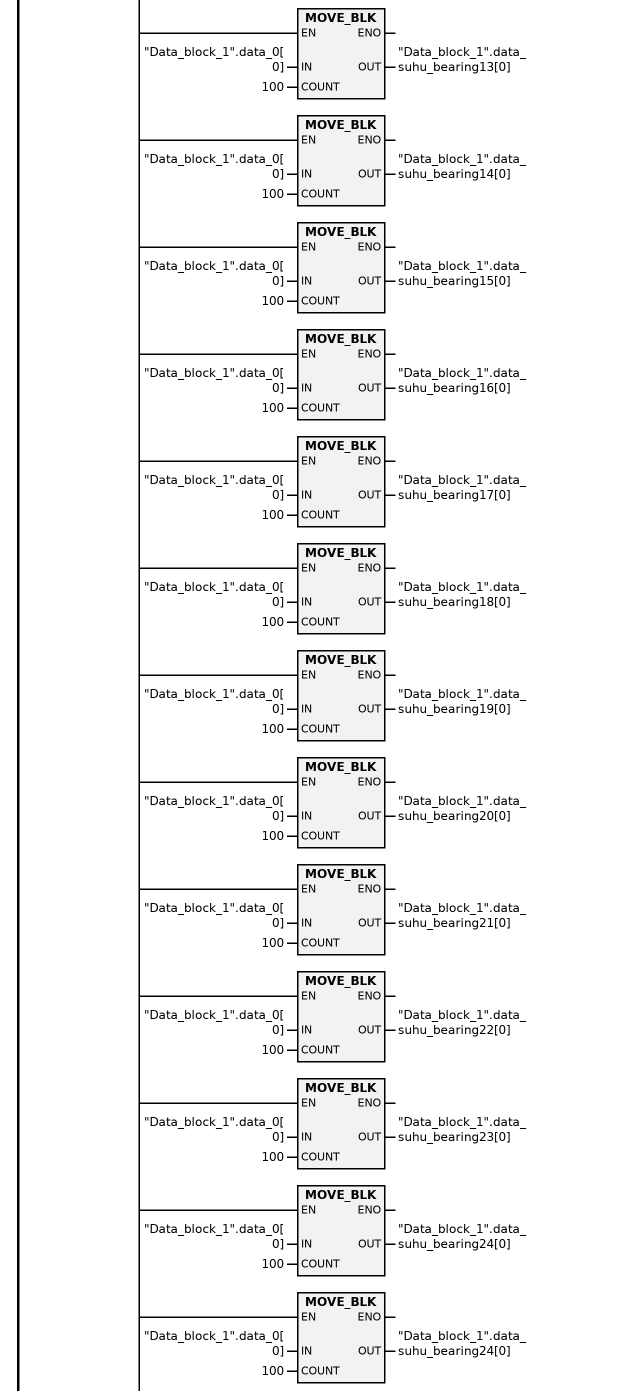
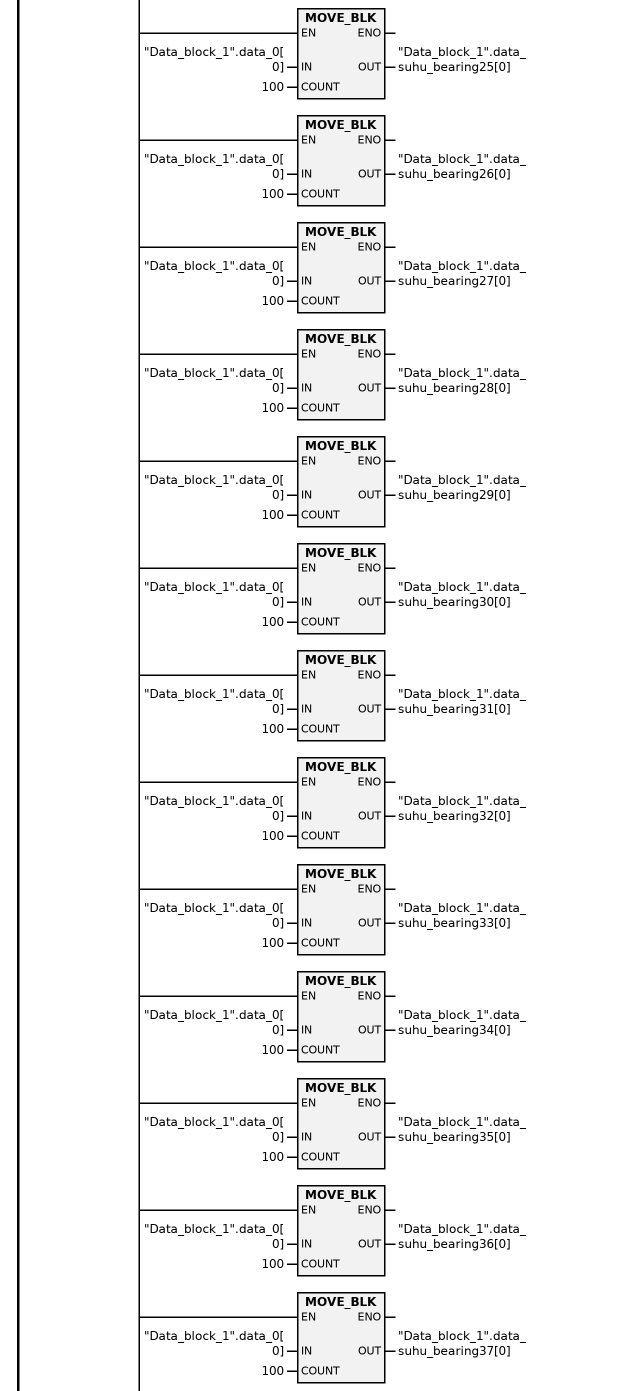
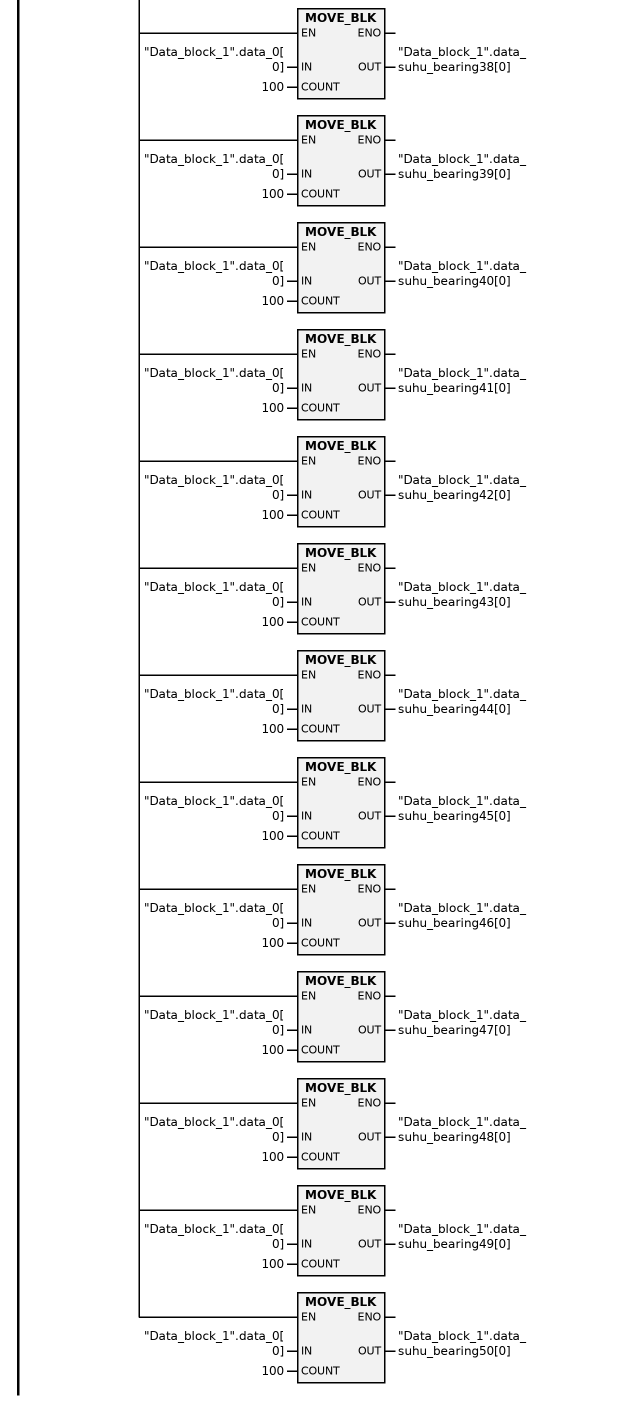
   #_w1 := "Data_block_1".Reset;
   IF #_w1 THEN
       MOVE_BLK(IN := "Data_block_1".data_0[0], COUNT := 100, OUT => "Data_block_1".data_suhu_bearing1[0]);
       MOVE_BLK(IN := "Data_block_1".data_0[0], COUNT := 100, OUT => "Data_block_1".data_suhu_bearing2[0]);
       MOVE_BLK(IN := "Data_block_1".data_0[0], COUNT := 100, OUT => "Data_block_1".data_suhu_bearing3[0]);
       MOVE_BLK(IN := "Data_block_1".data_0[0], COUNT := 100, OUT => "Data_block_1".data_suhu_bearing4[0]);
       MOVE_BLK(IN := "Data_block_1".data_0[0], COUNT := 100, OUT => "Data_block_1".data_suhu_bearing5[0]);
       MOVE_BLK(IN := "Data_block_1".data_0[0], COUNT := 100, OUT => "Data_block_1".data_suhu_bearing6[0]);
       MOVE_BLK(IN := "Data_block_1".data_0[0], COUNT := 100, OUT => "Data_block_1".data_suhu_bearing7[0]);
       MOVE_BLK(IN := "Data_block_1".data_0[0], COUNT := 100, OUT => "Data_block_1".data_suhu_bearing8[0]);
       MOVE_BLK(IN := "Data_block_1".data_0[0], COUNT := 100, OUT => "Data_block_1".data_suhu_bearing9[0]);
       MOVE_BLK(IN := "Data_block_1".data_0[0], COUNT := 100, OUT => "Data_block_1".data_suhu_bearing10[0]);
       MOVE_BLK(IN := "Data_block_1".data_0[0], COUNT := 100, OUT => "Data_block_1".data_suhu_bearing11[0]);
       MOVE_BLK(IN := "Data_block_1".data_0[0], COUNT := 100, OUT => "Data_block_1".data_suhu_bearing12[0]);
       MOVE_BLK(IN := "Data_block_1".data_0[0], COUNT := 100, OUT => "Data_block_1".data_suhu_bearing13[0]);
       MOVE_BLK(IN := "Data_block_1".data_0[0], COUNT := 100, OUT => "Data_block_1".data_suhu_bearing14[0]);
       MOVE_BLK(IN := "Data_block_1".data_0[0], COUNT := 100, OUT => "Data_block_1".data_suhu_bearing15[0]);
       MOVE_BLK(IN := "Data_block_1".data_0[0], COUNT := 100, OUT => "Data_block_1".data_suhu_bearing16[0]);
       MOVE_BLK(IN := "Data_block_1".data_0[0], COUNT := 100, OUT => "Data_block_1".data_suhu_bearing17[0]);
       MOVE_BLK(IN := "Data_block_1".data_0[0], COUNT := 100, OUT => "Data_block_1".data_suhu_bearing18[0]);
       MOVE_BLK(IN := "Data_block_1".data_0[0], COUNT := 100, OUT => "Data_block_1".data_suhu_bearing19[0]);
       MOVE_BLK(IN := "Data_block_1".data_0[0], COUNT := 100, OUT => "Data_block_1".data_suhu_bearing20[0]);
       MOVE_BLK(IN := "Data_block_1".data_0[0], COUNT := 100, OUT => "Data_block_1".data_suhu_bearing21[0]);
       MOVE_BLK(IN := "Data_block_1".data_0[0], COUNT := 100, OUT => "Data_block_1".data_suhu_bearing22[0]);
       MOVE_BLK(IN := "Data_block_1".data_0[0], COUNT := 100, OUT => "Data_block_1".data_suhu_bearing23[0]);
       MOVE_BLK(IN := "Data_block_1".data_0[0], COUNT := 100, OUT => "Data_block_1".data_suhu_bearing24[0]);
       MOVE_BLK(IN := "Data_block_1".data_0[0], COUNT := 100, OUT => "Data_block_1".data_suhu_bearing24[0]);
       MOVE_BLK(IN := "Data_block_1".data_0[0], COUNT := 100, OUT => "Data_block_1".data_suhu_bearing25[0]);
       MOVE_BLK(IN := "Data_block_1".data_0[0], COUNT := 100, OUT => "Data_block_1".data_suhu_bearing26[0]);
       MOVE_BLK(IN := "Data_block_1".data_0[0], COUNT := 100, OUT => "Data_block_1".data_suhu_bearing27[0]);
       MOVE_BLK(IN := "Data_block_1".data_0[0], COUNT := 100, OUT => "Data_block_1".data_suhu_bearing28[0]);
       MOVE_BLK(IN := "Data_block_1".data_0[0], COUNT := 100, OUT => "Data_block_1".data_suhu_bearing29[0]);
       MOVE_BLK(IN := "Data_block_1".data_0[0], COUNT := 100, OUT => "Data_block_1".data_suhu_bearing30[0]);
       MOVE_BLK(IN := "Data_block_1".data_0[0], COUNT := 100, OUT => "Data_block_1".data_suhu_bearing31[0]);
       MOVE_BLK(IN := "Data_block_1".data_0[0], COUNT := 100, OUT => "Data_block_1".data_suhu_bearing32[0]);
       MOVE_BLK(IN := "Data_block_1".data_0[0], COUNT := 100, OUT => "Data_block_1".data_suhu_bearing33[0]);
       MOVE_BLK(IN := "Data_block_1".data_0[0], COUNT := 100, OUT => "Data_block_1".data_suhu_bearing34[0]);
       MOVE_BLK(IN := "Data_block_1".data_0[0], COUNT := 100, OUT => "Data_block_1".data_suhu_bearing35[0]);
       MOVE_BLK(IN := "Data_block_1".data_0[0], COUNT := 100, OUT => "Data_block_1".data_suhu_bearing36[0]);
       MOVE_BLK(IN := "Data_block_1".data_0[0], COUNT := 100, OUT => "Data_block_1".data_suhu_bearing37[0]);
       MOVE_BLK(IN := "Data_block_1".data_0[0], COUNT := 100, OUT => "Data_block_1".data_suhu_bearing38[0]);
       MOVE_BLK(IN := "Data_block_1".data_0[0], COUNT := 100, OUT => "Data_block_1".data_suhu_bearing39[0]);
       MOVE_BLK(IN := "Data_block_1".data_0[0], COUNT := 100, OUT => "Data_block_1".data_suhu_bearing40[0]);
       MOVE_BLK(IN := "Data_block_1".data_0[0], COUNT := 100, OUT => "Data_block_1".data_suhu_bearing41[0]);
       MOVE_BLK(IN := "Data_block_1".data_0[0], COUNT := 100, OUT => "Data_block_1".data_suhu_bearing42[0]);
       MOVE_BLK(IN := "Data_block_1".data_0[0], COUNT := 100, OUT => "Data_block_1".data_suhu_bearing43[0]);
       MOVE_BLK(IN := "Data_block_1".data_0[0], COUNT := 100, OUT => "Data_block_1".data_suhu_bearing44[0]);
       MOVE_BLK(IN := "Data_block_1".data_0[0], COUNT := 100, OUT => "Data_block_1".data_suhu_bearing45[0]);
       MOVE_BLK(IN := "Data_block_1".data_0[0], COUNT := 100, OUT => "Data_block_1".data_suhu_bearing46[0]);
       MOVE_BLK(IN := "Data_block_1".data_0[0], COUNT := 100, OUT => "Data_block_1".data_suhu_bearing47[0]);
       MOVE_BLK(IN := "Data_block_1".data_0[0], COUNT := 100, OUT => "Data_block_1".data_suhu_bearing48[0]);
       MOVE_BLK(IN := "Data_block_1".data_0[0], COUNT := 100, OUT => "Data_block_1".data_suhu_bearing49[0]);
       MOVE_BLK(IN := "Data_block_1".data_0[0], COUNT := 100, OUT => "Data_block_1".data_suhu_bearing50[0]);
   END_IF;
END_REGION

REGION Network 24: Mengukur Suhu Roda (kiri ke kanan)
   // setelah sensor suhu aktif membaca
   // kemudian counter menghitung jumlah berapa kali sensor suhu mendeteksi suhu pada satu roda
   // 
   // apabila data sensor suhu yang terbaca(datasensor) tidak sama dengan nol maka data suhu yang terbaca(datasensor) dipindahkan ke array data suhu baru (data_baru1 untuk sebelah kanan) (data_baru2 untuk sebelah kiri)
   // data sensor terbaru dirubah jadi data baru
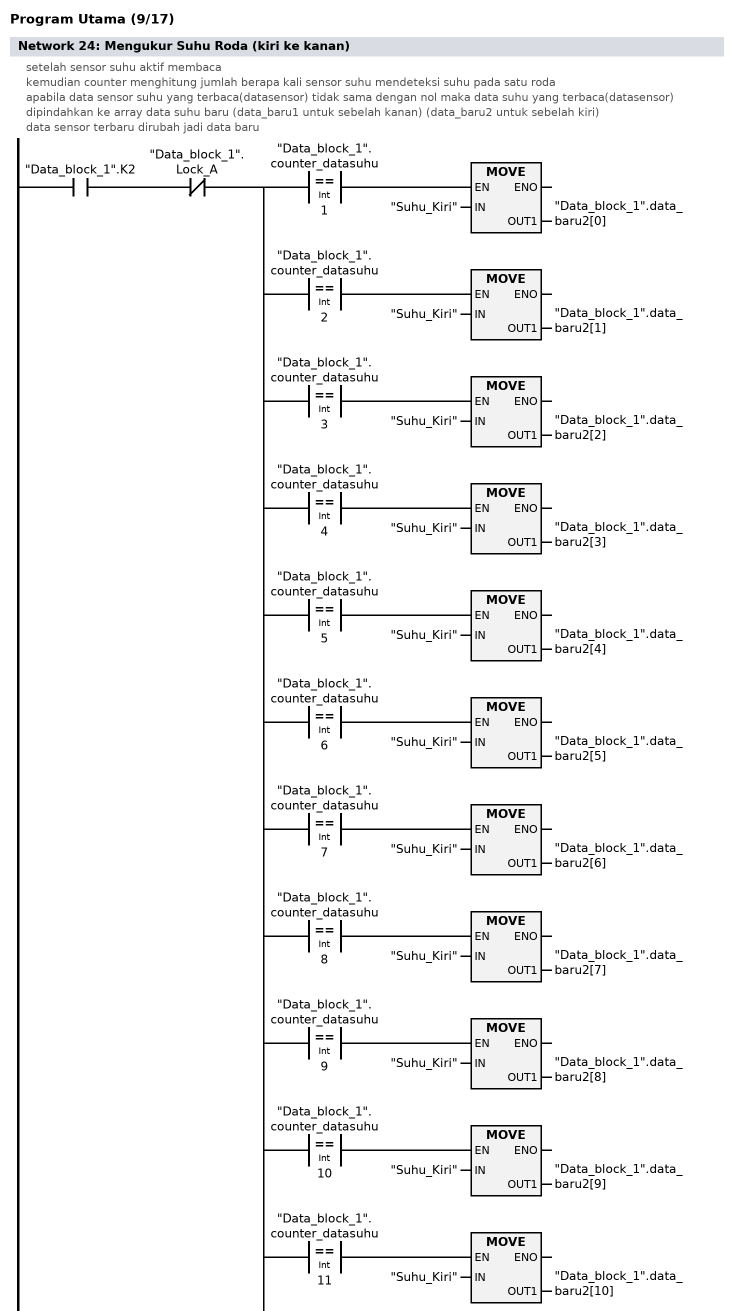
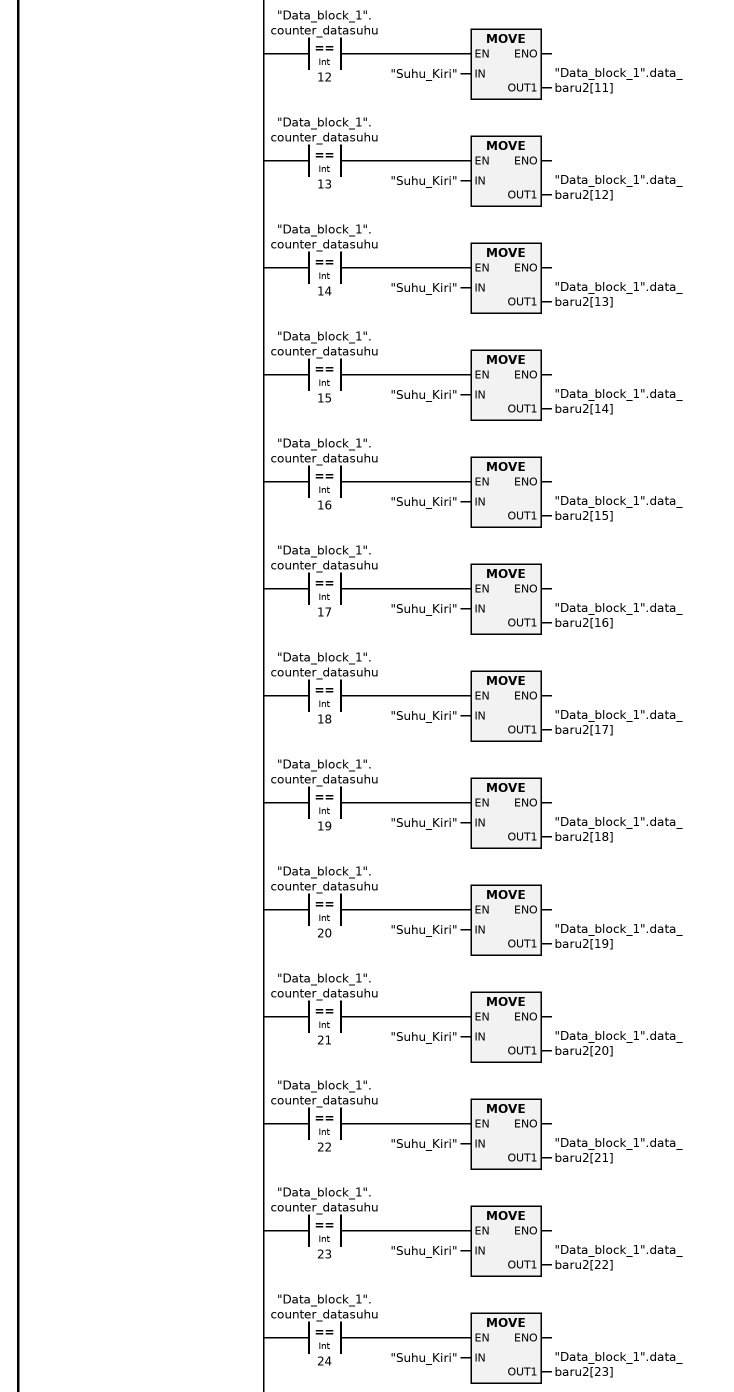
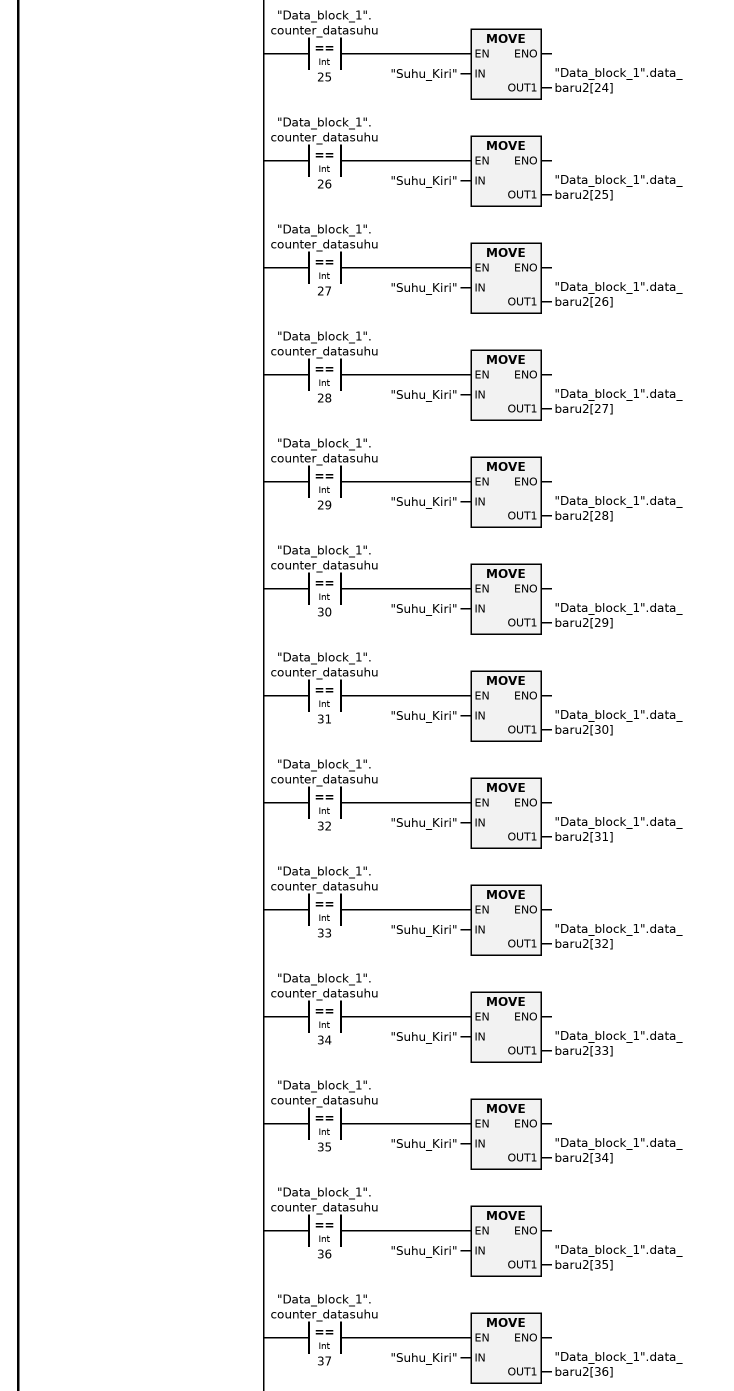
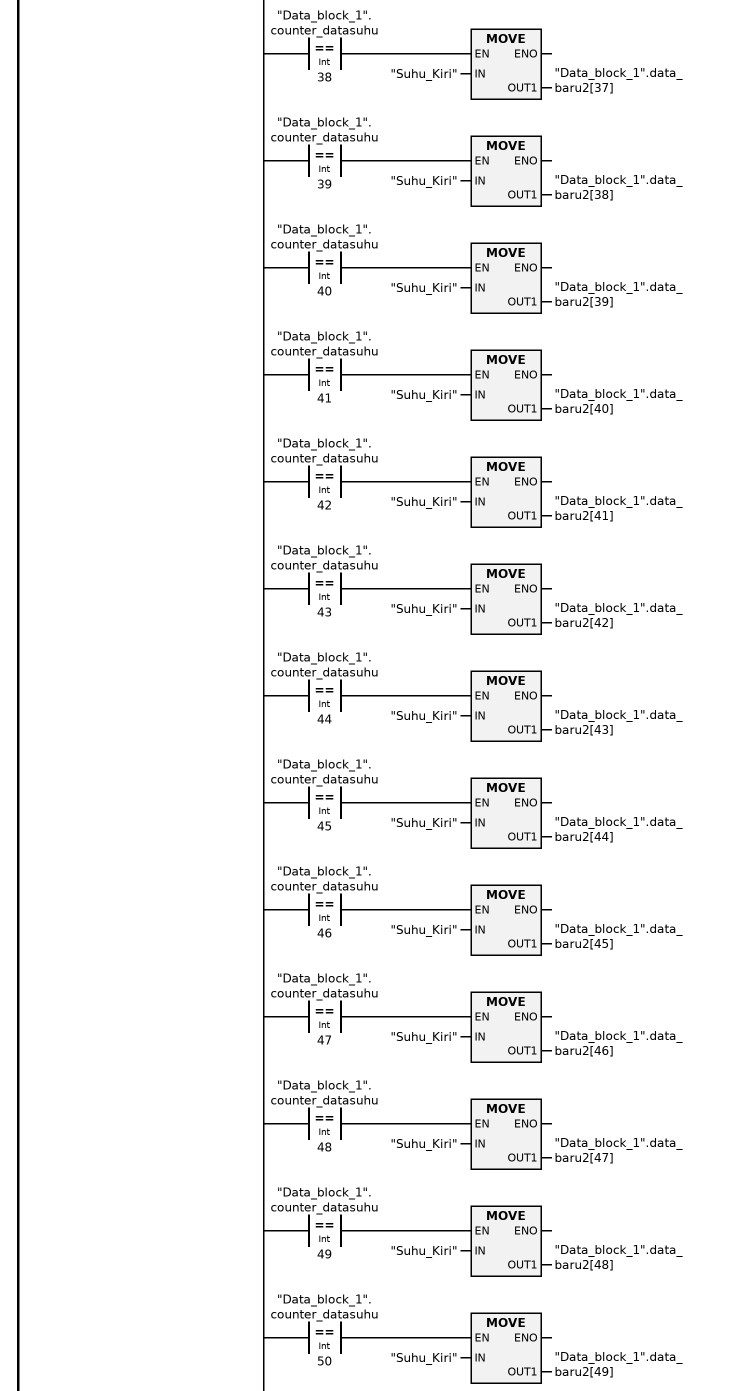
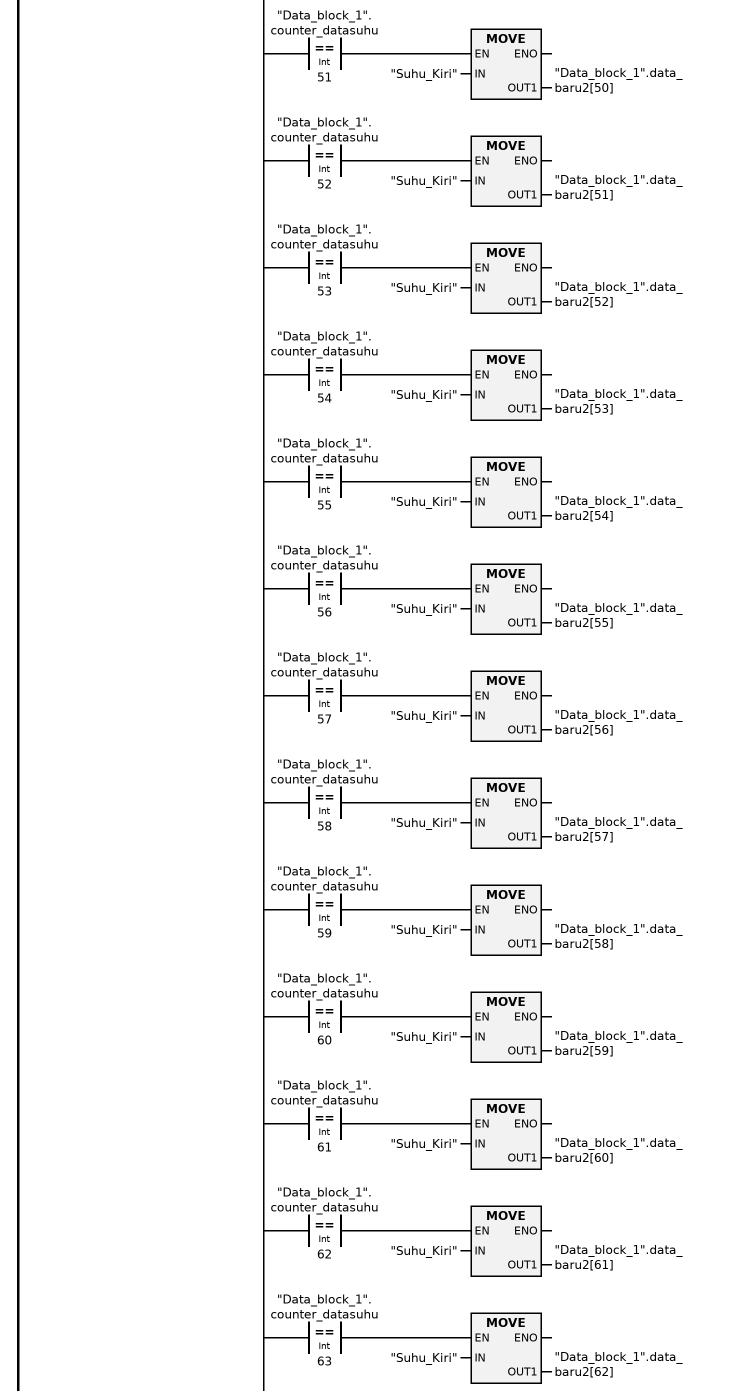
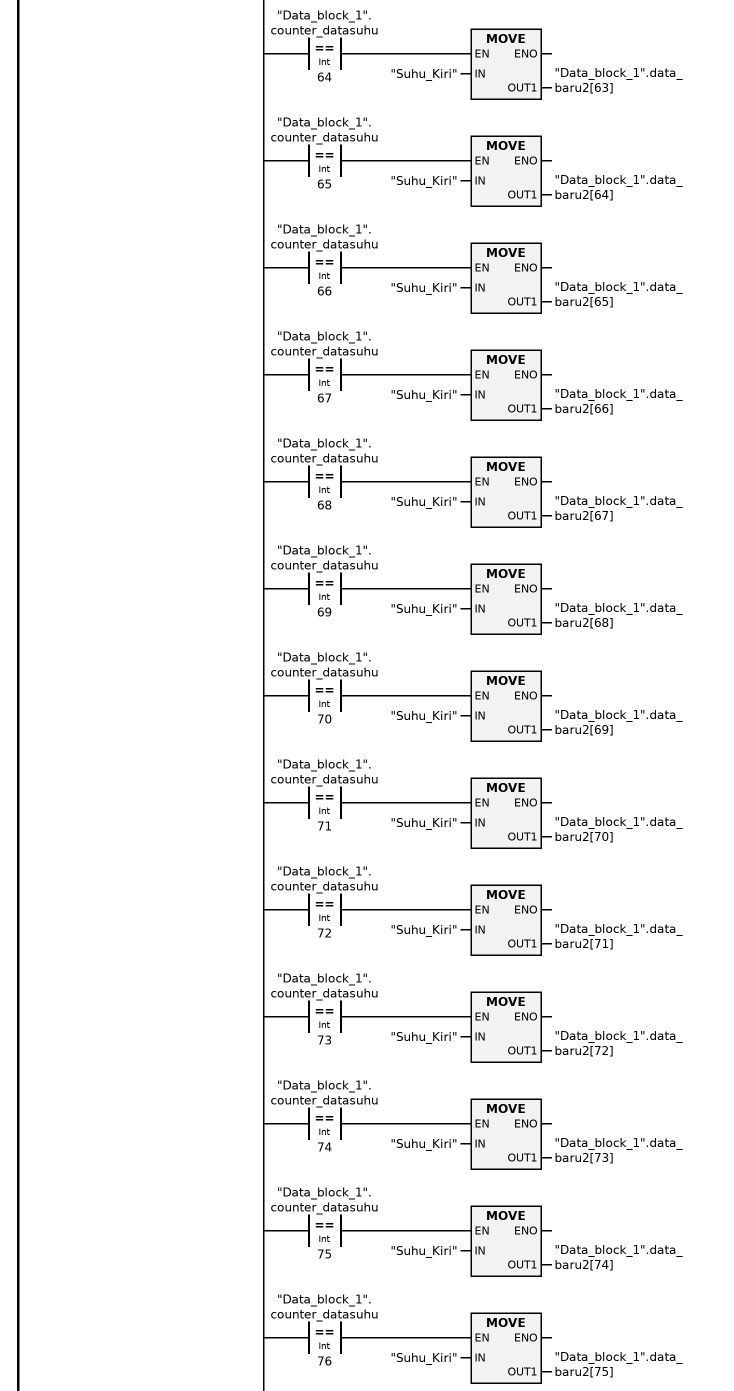
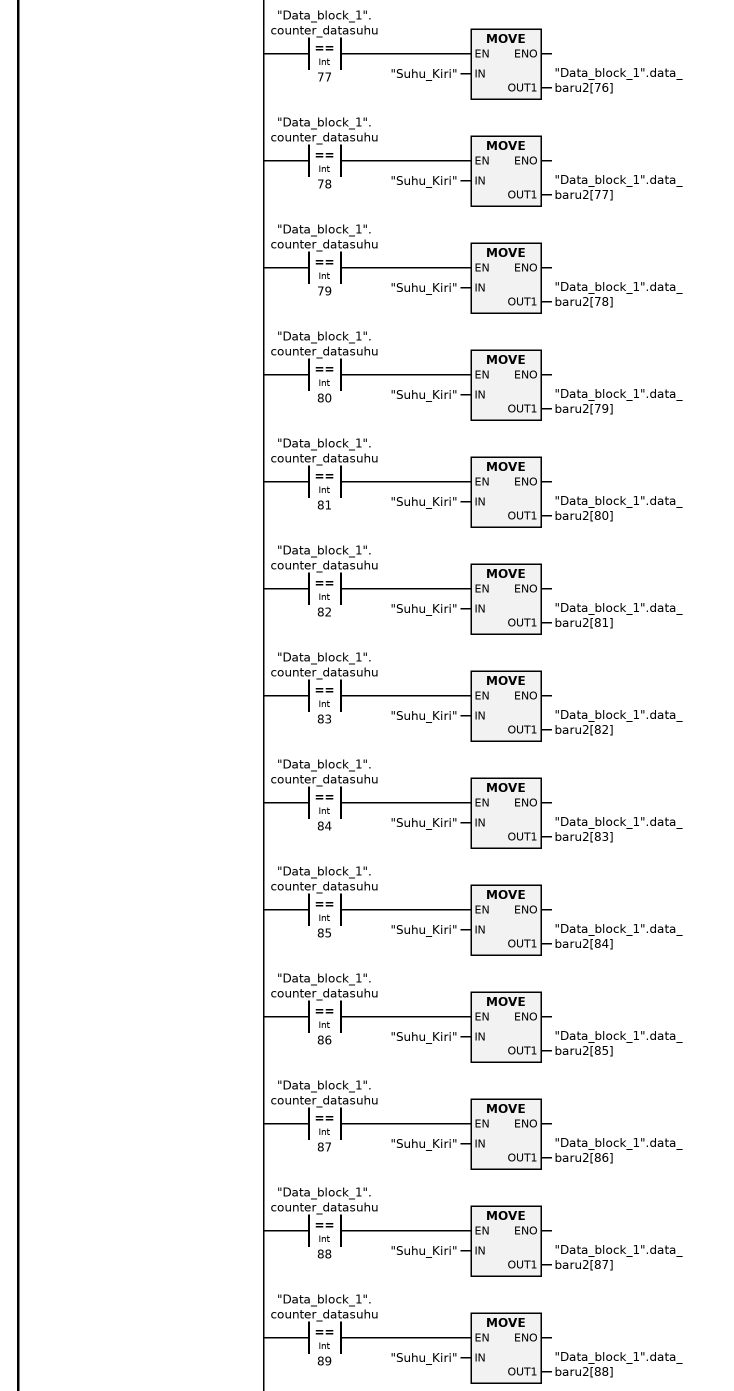
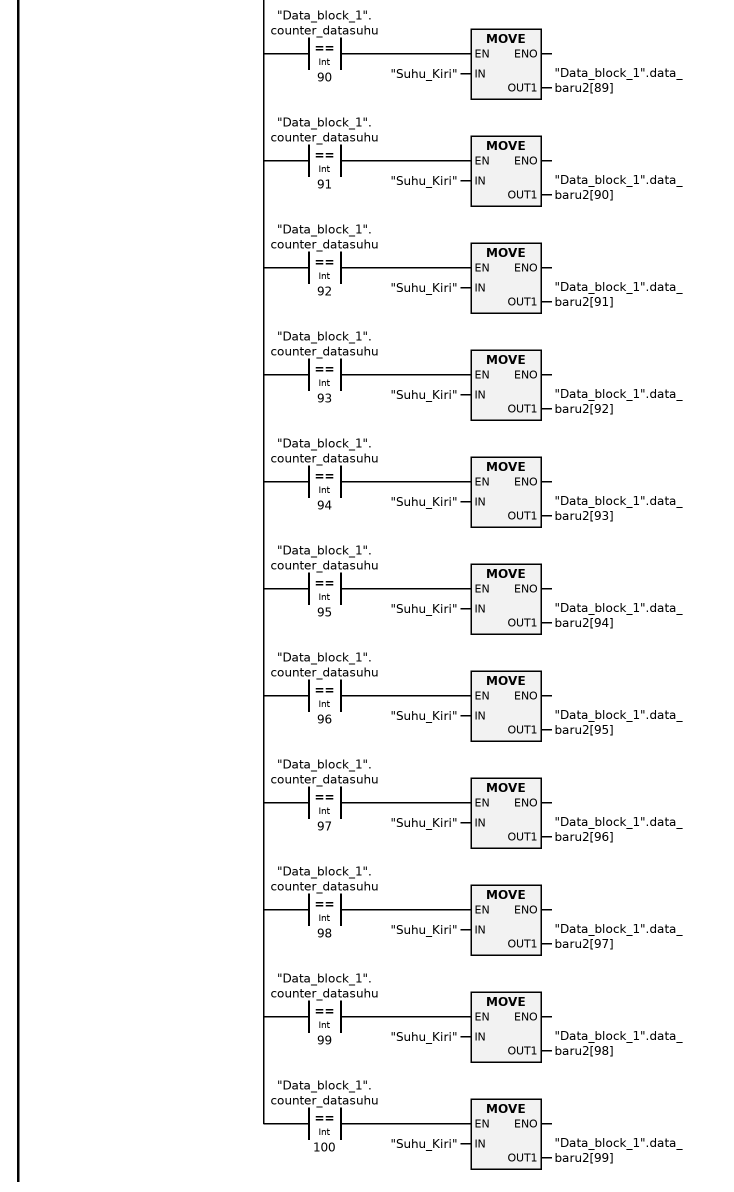
   RUNG wire#powerrail
      Contact( "Data_block_1".K2 )
      I_Contact( "Data_block_1".Lock_A )
      wire#w1
      { S7_Templates := "SrcType := Int" } EQ_Contact(in1 := "Data_block_1".counter_datasuhu, in2 := 1)
      Move(in := "Suhu_Kiri", out1 => "Data_block_1".data_baru2[0])
   END_RUNG
   RUNG wire#w1
      { S7_Templates := "SrcType := Int" } EQ_Contact(in1 := "Data_block_1".counter_datasuhu, in2 := 2)
      Move(in := "Suhu_Kiri", out1 => "Data_block_1".data_baru2[1])
   END_RUNG
   RUNG wire#w1
      { S7_Templates := "SrcType := Int" } EQ_Contact(in1 := "Data_block_1".counter_datasuhu, in2 := 3)
      Move(in := "Suhu_Kiri", out1 => "Data_block_1".data_baru2[2])
   END_RUNG
   RUNG wire#w1
      { S7_Templates := "SrcType := Int" } EQ_Contact(in1 := "Data_block_1".counter_datasuhu, in2 := 4)
      Move(in := "Suhu_Kiri", out1 => "Data_block_1".data_baru2[3])
   END_RUNG
   RUNG wire#w1
      { S7_Templates := "SrcType := Int" } EQ_Contact(in1 := "Data_block_1".counter_datasuhu, in2 := 5)
      Move(in := "Suhu_Kiri", out1 => "Data_block_1".data_baru2[4])
   END_RUNG
   RUNG wire#w1
      { S7_Templates := "SrcType := Int" } EQ_Contact(in1 := "Data_block_1".counter_datasuhu, in2 := 6)
      Move(in := "Suhu_Kiri", out1 => "Data_block_1".data_baru2[5])
   END_RUNG
   RUNG wire#w1
      { S7_Templates := "SrcType := Int" } EQ_Contact(in1 := "Data_block_1".counter_datasuhu, in2 := 7)
      Move(in := "Suhu_Kiri", out1 => "Data_block_1".data_baru2[6])
   END_RUNG
   RUNG wire#w1
      { S7_Templates := "SrcType := Int" } EQ_Contact(in1 := "Data_block_1".counter_datasuhu, in2 := 8)
      Move(in := "Suhu_Kiri", out1 => "Data_block_1".data_baru2[7])
   END_RUNG
   RUNG wire#w1
      { S7_Templates := "SrcType := Int" } EQ_Contact(in1 := "Data_block_1".counter_datasuhu, in2 := 9)
      Move(in := "Suhu_Kiri", out1 => "Data_block_1".data_baru2[8])
   END_RUNG
   RUNG wire#w1
      { S7_Templates := "SrcType := Int" } EQ_Contact(in1 := "Data_block_1".counter_datasuhu, in2 := 10)
      Move(in := "Suhu_Kiri", out1 => "Data_block_1".data_baru2[9])
   END_RUNG
   RUNG wire#w1
      { S7_Templates := "SrcType := Int" } EQ_Contact(in1 := "Data_block_1".counter_datasuhu, in2 := 11)
      Move(in := "Suhu_Kiri", out1 => "Data_block_1".data_baru2[10])
   END_RUNG
   RUNG wire#w1
      { S7_Templates := "SrcType := Int" } EQ_Contact(in1 := "Data_block_1".counter_datasuhu, in2 := 12)
      Move(in := "Suhu_Kiri", out1 => "Data_block_1".data_baru2[11])
   END_RUNG
   RUNG wire#w1
      { S7_Templates := "SrcType := Int" } EQ_Contact(in1 := "Data_block_1".counter_datasuhu, in2 := 13)
      Move(in := "Suhu_Kiri", out1 => "Data_block_1".data_baru2[12])
   END_RUNG
   RUNG wire#w1
      { S7_Templates := "SrcType := Int" } EQ_Contact(in1 := "Data_block_1".counter_datasuhu, in2 := 14)
      Move(in := "Suhu_Kiri", out1 => "Data_block_1".data_baru2[13])
   END_RUNG
   RUNG wire#w1
      { S7_Templates := "SrcType := Int" } EQ_Contact(in1 := "Data_block_1".counter_datasuhu, in2 := 15)
      Move(in := "Suhu_Kiri", out1 => "Data_block_1".data_baru2[14])
   END_RUNG
   RUNG wire#w1
      { S7_Templates := "SrcType := Int" } EQ_Contact(in1 := "Data_block_1".counter_datasuhu, in2 := 16)
      Move(in := "Suhu_Kiri", out1 => "Data_block_1".data_baru2[15])
   END_RUNG
   RUNG wire#w1
      { S7_Templates := "SrcType := Int" } EQ_Contact(in1 := "Data_block_1".counter_datasuhu, in2 := 17)
      Move(in := "Suhu_Kiri", out1 => "Data_block_1".data_baru2[16])
   END_RUNG
   RUNG wire#w1
      { S7_Templates := "SrcType := Int" } EQ_Contact(in1 := "Data_block_1".counter_datasuhu, in2 := 18)
      Move(in := "Suhu_Kiri", out1 => "Data_block_1".data_baru2[17])
   END_RUNG
   RUNG wire#w1
      { S7_Templates := "SrcType := Int" } EQ_Contact(in1 := "Data_block_1".counter_datasuhu, in2 := 19)
      Move(in := "Suhu_Kiri", out1 => "Data_block_1".data_baru2[18])
   END_RUNG
   RUNG wire#w1
      { S7_Templates := "SrcType := Int" } EQ_Contact(in1 := "Data_block_1".counter_datasuhu, in2 := 20)
      Move(in := "Suhu_Kiri", out1 => "Data_block_1".data_baru2[19])
   END_RUNG
   RUNG wire#w1
      { S7_Templates := "SrcType := Int" } EQ_Contact(in1 := "Data_block_1".counter_datasuhu, in2 := 21)
      Move(in := "Suhu_Kiri", out1 => "Data_block_1".data_baru2[20])
   END_RUNG
   RUNG wire#w1
      { S7_Templates := "SrcType := Int" } EQ_Contact(in1 := "Data_block_1".counter_datasuhu, in2 := 22)
      Move(in := "Suhu_Kiri", out1 => "Data_block_1".data_baru2[21])
   END_RUNG
   RUNG wire#w1
      { S7_Templates := "SrcType := Int" } EQ_Contact(in1 := "Data_block_1".counter_datasuhu, in2 := 23)
      Move(in := "Suhu_Kiri", out1 => "Data_block_1".data_baru2[22])
   END_RUNG
   RUNG wire#w1
      { S7_Templates := "SrcType := Int" } EQ_Contact(in1 := "Data_block_1".counter_datasuhu, in2 := 24)
      Move(in := "Suhu_Kiri", out1 => "Data_block_1".data_baru2[23])
   END_RUNG
   RUNG wire#w1
      { S7_Templates := "SrcType := Int" } EQ_Contact(in1 := "Data_block_1".counter_datasuhu, in2 := 25)
      Move(in := "Suhu_Kiri", out1 => "Data_block_1".data_baru2[24])
   END_RUNG
   RUNG wire#w1
      { S7_Templates := "SrcType := Int" } EQ_Contact(in1 := "Data_block_1".counter_datasuhu, in2 := 26)
      Move(in := "Suhu_Kiri", out1 => "Data_block_1".data_baru2[25])
   END_RUNG
   RUNG wire#w1
      { S7_Templates := "SrcType := Int" } EQ_Contact(in1 := "Data_block_1".counter_datasuhu, in2 := 27)
      Move(in := "Suhu_Kiri", out1 => "Data_block_1".data_baru2[26])
   END_RUNG
   RUNG wire#w1
      { S7_Templates := "SrcType := Int" } EQ_Contact(in1 := "Data_block_1".counter_datasuhu, in2 := 28)
      Move(in := "Suhu_Kiri", out1 => "Data_block_1".data_baru2[27])
   END_RUNG
   RUNG wire#w1
      { S7_Templates := "SrcType := Int" } EQ_Contact(in1 := "Data_block_1".counter_datasuhu, in2 := 29)
      Move(in := "Suhu_Kiri", out1 => "Data_block_1".data_baru2[28])
   END_RUNG
   RUNG wire#w1
      { S7_Templates := "SrcType := Int" } EQ_Contact(in1 := "Data_block_1".counter_datasuhu, in2 := 30)
      Move(in := "Suhu_Kiri", out1 => "Data_block_1".data_baru2[29])
   END_RUNG
   RUNG wire#w1
      { S7_Templates := "SrcType := Int" } EQ_Contact(in1 := "Data_block_1".counter_datasuhu, in2 := 31)
      Move(in := "Suhu_Kiri", out1 => "Data_block_1".data_baru2[30])
   END_RUNG
   RUNG wire#w1
      { S7_Templates := "SrcType := Int" } EQ_Contact(in1 := "Data_block_1".counter_datasuhu, in2 := 32)
      Move(in := "Suhu_Kiri", out1 => "Data_block_1".data_baru2[31])
   END_RUNG
   RUNG wire#w1
      { S7_Templates := "SrcType := Int" } EQ_Contact(in1 := "Data_block_1".counter_datasuhu, in2 := 33)
      Move(in := "Suhu_Kiri", out1 => "Data_block_1".data_baru2[32])
   END_RUNG
   RUNG wire#w1
      { S7_Templates := "SrcType := Int" } EQ_Contact(in1 := "Data_block_1".counter_datasuhu, in2 := 34)
      Move(in := "Suhu_Kiri", out1 => "Data_block_1".data_baru2[33])
   END_RUNG
   RUNG wire#w1
      { S7_Templates := "SrcType := Int" } EQ_Contact(in1 := "Data_block_1".counter_datasuhu, in2 := 35)
      Move(in := "Suhu_Kiri", out1 => "Data_block_1".data_baru2[34])
   END_RUNG
   RUNG wire#w1
      { S7_Templates := "SrcType := Int" } EQ_Contact(in1 := "Data_block_1".counter_datasuhu, in2 := 36)
      Move(in := "Suhu_Kiri", out1 => "Data_block_1".data_baru2[35])
   END_RUNG
   RUNG wire#w1
      { S7_Templates := "SrcType := Int" } EQ_Contact(in1 := "Data_block_1".counter_datasuhu, in2 := 37)
      Move(in := "Suhu_Kiri", out1 => "Data_block_1".data_baru2[36])
   END_RUNG
   RUNG wire#w1
      { S7_Templates := "SrcType := Int" } EQ_Contact(in1 := "Data_block_1".counter_datasuhu, in2 := 38)
      Move(in := "Suhu_Kiri", out1 => "Data_block_1".data_baru2[37])
   END_RUNG
   RUNG wire#w1
      { S7_Templates := "SrcType := Int" } EQ_Contact(in1 := "Data_block_1".counter_datasuhu, in2 := 39)
      Move(in := "Suhu_Kiri", out1 => "Data_block_1".data_baru2[38])
   END_RUNG
   RUNG wire#w1
      { S7_Templates := "SrcType := Int" } EQ_Contact(in1 := "Data_block_1".counter_datasuhu, in2 := 40)
      Move(in := "Suhu_Kiri", out1 => "Data_block_1".data_baru2[39])
   END_RUNG
   RUNG wire#w1
      { S7_Templates := "SrcType := Int" } EQ_Contact(in1 := "Data_block_1".counter_datasuhu, in2 := 41)
      Move(in := "Suhu_Kiri", out1 => "Data_block_1".data_baru2[40])
   END_RUNG
   RUNG wire#w1
      { S7_Templates := "SrcType := Int" } EQ_Contact(in1 := "Data_block_1".counter_datasuhu, in2 := 42)
      Move(in := "Suhu_Kiri", out1 => "Data_block_1".data_baru2[41])
   END_RUNG
   RUNG wire#w1
      { S7_Templates := "SrcType := Int" } EQ_Contact(in1 := "Data_block_1".counter_datasuhu, in2 := 43)
      Move(in := "Suhu_Kiri", out1 => "Data_block_1".data_baru2[42])
   END_RUNG
   RUNG wire#w1
      { S7_Templates := "SrcType := Int" } EQ_Contact(in1 := "Data_block_1".counter_datasuhu, in2 := 44)
      Move(in := "Suhu_Kiri", out1 => "Data_block_1".data_baru2[43])
   END_RUNG
   RUNG wire#w1
      { S7_Templates := "SrcType := Int" } EQ_Contact(in1 := "Data_block_1".counter_datasuhu, in2 := 45)
      Move(in := "Suhu_Kiri", out1 => "Data_block_1".data_baru2[44])
   END_RUNG
   RUNG wire#w1
      { S7_Templates := "SrcType := Int" } EQ_Contact(in1 := "Data_block_1".counter_datasuhu, in2 := 46)
      Move(in := "Suhu_Kiri", out1 => "Data_block_1".data_baru2[45])
   END_RUNG
   RUNG wire#w1
      { S7_Templates := "SrcType := Int" } EQ_Contact(in1 := "Data_block_1".counter_datasuhu, in2 := 47)
      Move(in := "Suhu_Kiri", out1 => "Data_block_1".data_baru2[46])
   END_RUNG
   RUNG wire#w1
      { S7_Templates := "SrcType := Int" } EQ_Contact(in1 := "Data_block_1".counter_datasuhu, in2 := 48)
      Move(in := "Suhu_Kiri", out1 => "Data_block_1".data_baru2[47])
   END_RUNG
   RUNG wire#w1
      { S7_Templates := "SrcType := Int" } EQ_Contact(in1 := "Data_block_1".counter_datasuhu, in2 := 49)
      Move(in := "Suhu_Kiri", out1 => "Data_block_1".data_baru2[48])
   END_RUNG
   RUNG wire#w1
      { S7_Templates := "SrcType := Int" } EQ_Contact(in1 := "Data_block_1".counter_datasuhu, in2 := 50)
      Move(in := "Suhu_Kiri", out1 => "Data_block_1".data_baru2[49])
   END_RUNG
   RUNG wire#w1
      { S7_Templates := "SrcType := Int" } EQ_Contact(in1 := "Data_block_1".counter_datasuhu, in2 := 51)
      Move(in := "Suhu_Kiri", out1 => "Data_block_1".data_baru2[50])
   END_RUNG
   RUNG wire#w1
      { S7_Templates := "SrcType := Int" } EQ_Contact(in1 := "Data_block_1".counter_datasuhu, in2 := 52)
      Move(in := "Suhu_Kiri", out1 => "Data_block_1".data_baru2[51])
   END_RUNG
   RUNG wire#w1
      { S7_Templates := "SrcType := Int" } EQ_Contact(in1 := "Data_block_1".counter_datasuhu, in2 := 53)
      Move(in := "Suhu_Kiri", out1 => "Data_block_1".data_baru2[52])
   END_RUNG
   RUNG wire#w1
      { S7_Templates := "SrcType := Int" } EQ_Contact(in1 := "Data_block_1".counter_datasuhu, in2 := 54)
      Move(in := "Suhu_Kiri", out1 => "Data_block_1".data_baru2[53])
   END_RUNG
   RUNG wire#w1
      { S7_Templates := "SrcType := Int" } EQ_Contact(in1 := "Data_block_1".counter_datasuhu, in2 := 55)
      Move(in := "Suhu_Kiri", out1 => "Data_block_1".data_baru2[54])
   END_RUNG
   RUNG wire#w1
      { S7_Templates := "SrcType := Int" } EQ_Contact(in1 := "Data_block_1".counter_datasuhu, in2 := 56)
      Move(in := "Suhu_Kiri", out1 => "Data_block_1".data_baru2[55])
   END_RUNG
   RUNG wire#w1
      { S7_Templates := "SrcType := Int" } EQ_Contact(in1 := "Data_block_1".counter_datasuhu, in2 := 57)
      Move(in := "Suhu_Kiri", out1 => "Data_block_1".data_baru2[56])
   END_RUNG
   RUNG wire#w1
      { S7_Templates := "SrcType := Int" } EQ_Contact(in1 := "Data_block_1".counter_datasuhu, in2 := 58)
      Move(in := "Suhu_Kiri", out1 => "Data_block_1".data_baru2[57])
   END_RUNG
   RUNG wire#w1
      { S7_Templates := "SrcType := Int" } EQ_Contact(in1 := "Data_block_1".counter_datasuhu, in2 := 59)
      Move(in := "Suhu_Kiri", out1 => "Data_block_1".data_baru2[58])
   END_RUNG
   RUNG wire#w1
      { S7_Templates := "SrcType := Int" } EQ_Contact(in1 := "Data_block_1".counter_datasuhu, in2 := 60)
      Move(in := "Suhu_Kiri", out1 => "Data_block_1".data_baru2[59])
   END_RUNG
   RUNG wire#w1
      { S7_Templates := "SrcType := Int" } EQ_Contact(in1 := "Data_block_1".counter_datasuhu, in2 := 61)
      Move(in := "Suhu_Kiri", out1 => "Data_block_1".data_baru2[60])
   END_RUNG
   RUNG wire#w1
      { S7_Templates := "SrcType := Int" } EQ_Contact(in1 := "Data_block_1".counter_datasuhu, in2 := 62)
      Move(in := "Suhu_Kiri", out1 => "Data_block_1".data_baru2[61])
   END_RUNG
   RUNG wire#w1
      { S7_Templates := "SrcType := Int" } EQ_Contact(in1 := "Data_block_1".counter_datasuhu, in2 := 63)
      Move(in := "Suhu_Kiri", out1 => "Data_block_1".data_baru2[62])
   END_RUNG
   RUNG wire#w1
      { S7_Templates := "SrcType := Int" } EQ_Contact(in1 := "Data_block_1".counter_datasuhu, in2 := 64)
      Move(in := "Suhu_Kiri", out1 => "Data_block_1".data_baru2[63])
   END_RUNG
   RUNG wire#w1
      { S7_Templates := "SrcType := Int" } EQ_Contact(in1 := "Data_block_1".counter_datasuhu, in2 := 65)
      Move(in := "Suhu_Kiri", out1 => "Data_block_1".data_baru2[64])
   END_RUNG
   RUNG wire#w1
      { S7_Templates := "SrcType := Int" } EQ_Contact(in1 := "Data_block_1".counter_datasuhu, in2 := 66)
      Move(in := "Suhu_Kiri", out1 => "Data_block_1".data_baru2[65])
   END_RUNG
   RUNG wire#w1
      { S7_Templates := "SrcType := Int" } EQ_Contact(in1 := "Data_block_1".counter_datasuhu, in2 := 67)
      Move(in := "Suhu_Kiri", out1 => "Data_block_1".data_baru2[66])
   END_RUNG
   RUNG wire#w1
      { S7_Templates := "SrcType := Int" } EQ_Contact(in1 := "Data_block_1".counter_datasuhu, in2 := 68)
      Move(in := "Suhu_Kiri", out1 => "Data_block_1".data_baru2[67])
   END_RUNG
   RUNG wire#w1
      { S7_Templates := "SrcType := Int" } EQ_Contact(in1 := "Data_block_1".counter_datasuhu, in2 := 69)
      Move(in := "Suhu_Kiri", out1 => "Data_block_1".data_baru2[68])
   END_RUNG
   RUNG wire#w1
      { S7_Templates := "SrcType := Int" } EQ_Contact(in1 := "Data_block_1".counter_datasuhu, in2 := 70)
      Move(in := "Suhu_Kiri", out1 => "Data_block_1".data_baru2[69])
   END_RUNG
   RUNG wire#w1
      { S7_Templates := "SrcType := Int" } EQ_Contact(in1 := "Data_block_1".counter_datasuhu, in2 := 71)
      Move(in := "Suhu_Kiri", out1 => "Data_block_1".data_baru2[70])
   END_RUNG
   RUNG wire#w1
      { S7_Templates := "SrcType := Int" } EQ_Contact(in1 := "Data_block_1".counter_datasuhu, in2 := 72)
      Move(in := "Suhu_Kiri", out1 => "Data_block_1".data_baru2[71])
   END_RUNG
   RUNG wire#w1
      { S7_Templates := "SrcType := Int" } EQ_Contact(in1 := "Data_block_1".counter_datasuhu, in2 := 73)
      Move(in := "Suhu_Kiri", out1 => "Data_block_1".data_baru2[72])
   END_RUNG
   RUNG wire#w1
      { S7_Templates := "SrcType := Int" } EQ_Contact(in1 := "Data_block_1".counter_datasuhu, in2 := 74)
      Move(in := "Suhu_Kiri", out1 => "Data_block_1".data_baru2[73])
   END_RUNG
   RUNG wire#w1
      { S7_Templates := "SrcType := Int" } EQ_Contact(in1 := "Data_block_1".counter_datasuhu, in2 := 75)
      Move(in := "Suhu_Kiri", out1 => "Data_block_1".data_baru2[74])
   END_RUNG
   RUNG wire#w1
      { S7_Templates := "SrcType := Int" } EQ_Contact(in1 := "Data_block_1".counter_datasuhu, in2 := 76)
      Move(in := "Suhu_Kiri", out1 => "Data_block_1".data_baru2[75])
   END_RUNG
   RUNG wire#w1
      { S7_Templates := "SrcType := Int" } EQ_Contact(in1 := "Data_block_1".counter_datasuhu, in2 := 77)
      Move(in := "Suhu_Kiri", out1 => "Data_block_1".data_baru2[76])
   END_RUNG
   RUNG wire#w1
      { S7_Templates := "SrcType := Int" } EQ_Contact(in1 := "Data_block_1".counter_datasuhu, in2 := 78)
      Move(in := "Suhu_Kiri", out1 => "Data_block_1".data_baru2[77])
   END_RUNG
   RUNG wire#w1
      { S7_Templates := "SrcType := Int" } EQ_Contact(in1 := "Data_block_1".counter_datasuhu, in2 := 79)
      Move(in := "Suhu_Kiri", out1 => "Data_block_1".data_baru2[78])
   END_RUNG
   RUNG wire#w1
      { S7_Templates := "SrcType := Int" } EQ_Contact(in1 := "Data_block_1".counter_datasuhu, in2 := 80)
      Move(in := "Suhu_Kiri", out1 => "Data_block_1".data_baru2[79])
   END_RUNG
   RUNG wire#w1
      { S7_Templates := "SrcType := Int" } EQ_Contact(in1 := "Data_block_1".counter_datasuhu, in2 := 81)
      Move(in := "Suhu_Kiri", out1 => "Data_block_1".data_baru2[80])
   END_RUNG
   RUNG wire#w1
      { S7_Templates := "SrcType := Int" } EQ_Contact(in1 := "Data_block_1".counter_datasuhu, in2 := 82)
      Move(in := "Suhu_Kiri", out1 => "Data_block_1".data_baru2[81])
   END_RUNG
   RUNG wire#w1
      { S7_Templates := "SrcType := Int" } EQ_Contact(in1 := "Data_block_1".counter_datasuhu, in2 := 83)
      Move(in := "Suhu_Kiri", out1 => "Data_block_1".data_baru2[82])
   END_RUNG
   RUNG wire#w1
      { S7_Templates := "SrcType := Int" } EQ_Contact(in1 := "Data_block_1".counter_datasuhu, in2 := 84)
      Move(in := "Suhu_Kiri", out1 => "Data_block_1".data_baru2[83])
   END_RUNG
   RUNG wire#w1
      { S7_Templates := "SrcType := Int" } EQ_Contact(in1 := "Data_block_1".counter_datasuhu, in2 := 85)
      Move(in := "Suhu_Kiri", out1 => "Data_block_1".data_baru2[84])
   END_RUNG
   RUNG wire#w1
      { S7_Templates := "SrcType := Int" } EQ_Contact(in1 := "Data_block_1".counter_datasuhu, in2 := 86)
      Move(in := "Suhu_Kiri", out1 => "Data_block_1".data_baru2[85])
   END_RUNG
   RUNG wire#w1
      { S7_Templates := "SrcType := Int" } EQ_Contact(in1 := "Data_block_1".counter_datasuhu, in2 := 87)
      Move(in := "Suhu_Kiri", out1 => "Data_block_1".data_baru2[86])
   END_RUNG
   RUNG wire#w1
      { S7_Templates := "SrcType := Int" } EQ_Contact(in1 := "Data_block_1".counter_datasuhu, in2 := 88)
      Move(in := "Suhu_Kiri", out1 => "Data_block_1".data_baru2[87])
   END_RUNG
   RUNG wire#w1
      { S7_Templates := "SrcType := Int" } EQ_Contact(in1 := "Data_block_1".counter_datasuhu, in2 := 89)
      Move(in := "Suhu_Kiri", out1 => "Data_block_1".data_baru2[88])
   END_RUNG
   RUNG wire#w1
      { S7_Templates := "SrcType := Int" } EQ_Contact(in1 := "Data_block_1".counter_datasuhu, in2 := 90)
      Move(in := "Suhu_Kiri", out1 => "Data_block_1".data_baru2[89])
   END_RUNG
   RUNG wire#w1
      { S7_Templates := "SrcType := Int" } EQ_Contact(in1 := "Data_block_1".counter_datasuhu, in2 := 91)
      Move(in := "Suhu_Kiri", out1 => "Data_block_1".data_baru2[90])
   END_RUNG
   RUNG wire#w1
      { S7_Templates := "SrcType := Int" } EQ_Contact(in1 := "Data_block_1".counter_datasuhu, in2 := 92)
      Move(in := "Suhu_Kiri", out1 => "Data_block_1".data_baru2[91])
   END_RUNG
   RUNG wire#w1
      { S7_Templates := "SrcType := Int" } EQ_Contact(in1 := "Data_block_1".counter_datasuhu, in2 := 93)
      Move(in := "Suhu_Kiri", out1 => "Data_block_1".data_baru2[92])
   END_RUNG
   RUNG wire#w1
      { S7_Templates := "SrcType := Int" } EQ_Contact(in1 := "Data_block_1".counter_datasuhu, in2 := 94)
      Move(in := "Suhu_Kiri", out1 => "Data_block_1".data_baru2[93])
   END_RUNG
   RUNG wire#w1
      { S7_Templates := "SrcType := Int" } EQ_Contact(in1 := "Data_block_1".counter_datasuhu, in2 := 95)
      Move(in := "Suhu_Kiri", out1 => "Data_block_1".data_baru2[94])
   END_RUNG
   RUNG wire#w1
      { S7_Templates := "SrcType := Int" } EQ_Contact(in1 := "Data_block_1".counter_datasuhu, in2 := 96)
      Move(in := "Suhu_Kiri", out1 => "Data_block_1".data_baru2[95])
   END_RUNG
   RUNG wire#w1
      { S7_Templates := "SrcType := Int" } EQ_Contact(in1 := "Data_block_1".counter_datasuhu, in2 := 97)
      Move(in := "Suhu_Kiri", out1 => "Data_block_1".data_baru2[96])
   END_RUNG
   RUNG wire#w1
      { S7_Templates := "SrcType := Int" } EQ_Contact(in1 := "Data_block_1".counter_datasuhu, in2 := 98)
      Move(in := "Suhu_Kiri", out1 => "Data_block_1".data_baru2[97])
   END_RUNG
   RUNG wire#w1
      { S7_Templates := "SrcType := Int" } EQ_Contact(in1 := "Data_block_1".counter_datasuhu, in2 := 99)
      Move(in := "Suhu_Kiri", out1 => "Data_block_1".data_baru2[98])
   END_RUNG
   RUNG wire#w1
      { S7_Templates := "SrcType := Int" } EQ_Contact(in1 := "Data_block_1".counter_datasuhu, in2 := 100)
      Move(in := "Suhu_Kiri", out1 => "Data_block_1".data_baru2[99])
   END_RUNG
   // the same network as SCL:
   #_w1 := "Data_block_1".K2 AND NOT "Data_block_1".Lock_A;
   IF #_w1 AND ("Data_block_1".counter_datasuhu = 1) THEN
       "Data_block_1".data_baru2[0] := "Suhu_Kiri";
   END_IF;
   IF #_w1 AND ("Data_block_1".counter_datasuhu = 2) THEN
       "Data_block_1".data_baru2[1] := "Suhu_Kiri";
   END_IF;
   IF #_w1 AND ("Data_block_1".counter_datasuhu = 3) THEN
       "Data_block_1".data_baru2[2] := "Suhu_Kiri";
   END_IF;
   IF #_w1 AND ("Data_block_1".counter_datasuhu = 4) THEN
       "Data_block_1".data_baru2[3] := "Suhu_Kiri";
   END_IF;
   IF #_w1 AND ("Data_block_1".counter_datasuhu = 5) THEN
       "Data_block_1".data_baru2[4] := "Suhu_Kiri";
   END_IF;
   IF #_w1 AND ("Data_block_1".counter_datasuhu = 6) THEN
       "Data_block_1".data_baru2[5] := "Suhu_Kiri";
   END_IF;
   IF #_w1 AND ("Data_block_1".counter_datasuhu = 7) THEN
       "Data_block_1".data_baru2[6] := "Suhu_Kiri";
   END_IF;
   IF #_w1 AND ("Data_block_1".counter_datasuhu = 8) THEN
       "Data_block_1".data_baru2[7] := "Suhu_Kiri";
   END_IF;
   IF #_w1 AND ("Data_block_1".counter_datasuhu = 9) THEN
       "Data_block_1".data_baru2[8] := "Suhu_Kiri";
   END_IF;
   IF #_w1 AND ("Data_block_1".counter_datasuhu = 10) THEN
       "Data_block_1".data_baru2[9] := "Suhu_Kiri";
   END_IF;
   IF #_w1 AND ("Data_block_1".counter_datasuhu = 11) THEN
       "Data_block_1".data_baru2[10] := "Suhu_Kiri";
   END_IF;
   IF #_w1 AND ("Data_block_1".counter_datasuhu = 12) THEN
       "Data_block_1".data_baru2[11] := "Suhu_Kiri";
   END_IF;
   IF #_w1 AND ("Data_block_1".counter_datasuhu = 13) THEN
       "Data_block_1".data_baru2[12] := "Suhu_Kiri";
   END_IF;
   IF #_w1 AND ("Data_block_1".counter_datasuhu = 14) THEN
       "Data_block_1".data_baru2[13] := "Suhu_Kiri";
   END_IF;
   IF #_w1 AND ("Data_block_1".counter_datasuhu = 15) THEN
       "Data_block_1".data_baru2[14] := "Suhu_Kiri";
   END_IF;
   IF #_w1 AND ("Data_block_1".counter_datasuhu = 16) THEN
       "Data_block_1".data_baru2[15] := "Suhu_Kiri";
   END_IF;
   IF #_w1 AND ("Data_block_1".counter_datasuhu = 17) THEN
       "Data_block_1".data_baru2[16] := "Suhu_Kiri";
   END_IF;
   IF #_w1 AND ("Data_block_1".counter_datasuhu = 18) THEN
       "Data_block_1".data_baru2[17] := "Suhu_Kiri";
   END_IF;
   IF #_w1 AND ("Data_block_1".counter_datasuhu = 19) THEN
       "Data_block_1".data_baru2[18] := "Suhu_Kiri";
   END_IF;
   IF #_w1 AND ("Data_block_1".counter_datasuhu = 20) THEN
       "Data_block_1".data_baru2[19] := "Suhu_Kiri";
   END_IF;
   IF #_w1 AND ("Data_block_1".counter_datasuhu = 21) THEN
       "Data_block_1".data_baru2[20] := "Suhu_Kiri";
   END_IF;
   IF #_w1 AND ("Data_block_1".counter_datasuhu = 22) THEN
       "Data_block_1".data_baru2[21] := "Suhu_Kiri";
   END_IF;
   IF #_w1 AND ("Data_block_1".counter_datasuhu = 23) THEN
       "Data_block_1".data_baru2[22] := "Suhu_Kiri";
   END_IF;
   IF #_w1 AND ("Data_block_1".counter_datasuhu = 24) THEN
       "Data_block_1".data_baru2[23] := "Suhu_Kiri";
   END_IF;
   IF #_w1 AND ("Data_block_1".counter_datasuhu = 25) THEN
       "Data_block_1".data_baru2[24] := "Suhu_Kiri";
   END_IF;
   IF #_w1 AND ("Data_block_1".counter_datasuhu = 26) THEN
       "Data_block_1".data_baru2[25] := "Suhu_Kiri";
   END_IF;
   IF #_w1 AND ("Data_block_1".counter_datasuhu = 27) THEN
       "Data_block_1".data_baru2[26] := "Suhu_Kiri";
   END_IF;
   IF #_w1 AND ("Data_block_1".counter_datasuhu = 28) THEN
       "Data_block_1".data_baru2[27] := "Suhu_Kiri";
   END_IF;
   IF #_w1 AND ("Data_block_1".counter_datasuhu = 29) THEN
       "Data_block_1".data_baru2[28] := "Suhu_Kiri";
   END_IF;
   IF #_w1 AND ("Data_block_1".counter_datasuhu = 30) THEN
       "Data_block_1".data_baru2[29] := "Suhu_Kiri";
   END_IF;
   IF #_w1 AND ("Data_block_1".counter_datasuhu = 31) THEN
       "Data_block_1".data_baru2[30] := "Suhu_Kiri";
   END_IF;
   IF #_w1 AND ("Data_block_1".counter_datasuhu = 32) THEN
       "Data_block_1".data_baru2[31] := "Suhu_Kiri";
   END_IF;
   IF #_w1 AND ("Data_block_1".counter_datasuhu = 33) THEN
       "Data_block_1".data_baru2[32] := "Suhu_Kiri";
   END_IF;
   IF #_w1 AND ("Data_block_1".counter_datasuhu = 34) THEN
       "Data_block_1".data_baru2[33] := "Suhu_Kiri";
   END_IF;
   IF #_w1 AND ("Data_block_1".counter_datasuhu = 35) THEN
       "Data_block_1".data_baru2[34] := "Suhu_Kiri";
   END_IF;
   IF #_w1 AND ("Data_block_1".counter_datasuhu = 36) THEN
       "Data_block_1".data_baru2[35] := "Suhu_Kiri";
   END_IF;
   IF #_w1 AND ("Data_block_1".counter_datasuhu = 37) THEN
       "Data_block_1".data_baru2[36] := "Suhu_Kiri";
   END_IF;
   IF #_w1 AND ("Data_block_1".counter_datasuhu = 38) THEN
       "Data_block_1".data_baru2[37] := "Suhu_Kiri";
   END_IF;
   IF #_w1 AND ("Data_block_1".counter_datasuhu = 39) THEN
       "Data_block_1".data_baru2[38] := "Suhu_Kiri";
   END_IF;
   IF #_w1 AND ("Data_block_1".counter_datasuhu = 40) THEN
       "Data_block_1".data_baru2[39] := "Suhu_Kiri";
   END_IF;
   IF #_w1 AND ("Data_block_1".counter_datasuhu = 41) THEN
       "Data_block_1".data_baru2[40] := "Suhu_Kiri";
   END_IF;
   IF #_w1 AND ("Data_block_1".counter_datasuhu = 42) THEN
       "Data_block_1".data_baru2[41] := "Suhu_Kiri";
   END_IF;
   IF #_w1 AND ("Data_block_1".counter_datasuhu = 43) THEN
       "Data_block_1".data_baru2[42] := "Suhu_Kiri";
   END_IF;
   IF #_w1 AND ("Data_block_1".counter_datasuhu = 44) THEN
       "Data_block_1".data_baru2[43] := "Suhu_Kiri";
   END_IF;
   IF #_w1 AND ("Data_block_1".counter_datasuhu = 45) THEN
       "Data_block_1".data_baru2[44] := "Suhu_Kiri";
   END_IF;
   IF #_w1 AND ("Data_block_1".counter_datasuhu = 46) THEN
       "Data_block_1".data_baru2[45] := "Suhu_Kiri";
   END_IF;
   IF #_w1 AND ("Data_block_1".counter_datasuhu = 47) THEN
       "Data_block_1".data_baru2[46] := "Suhu_Kiri";
   END_IF;
   IF #_w1 AND ("Data_block_1".counter_datasuhu = 48) THEN
       "Data_block_1".data_baru2[47] := "Suhu_Kiri";
   END_IF;
   IF #_w1 AND ("Data_block_1".counter_datasuhu = 49) THEN
       "Data_block_1".data_baru2[48] := "Suhu_Kiri";
   END_IF;
   IF #_w1 AND ("Data_block_1".counter_datasuhu = 50) THEN
       "Data_block_1".data_baru2[49] := "Suhu_Kiri";
   END_IF;
   IF #_w1 AND ("Data_block_1".counter_datasuhu = 51) THEN
       "Data_block_1".data_baru2[50] := "Suhu_Kiri";
   END_IF;
   IF #_w1 AND ("Data_block_1".counter_datasuhu = 52) THEN
       "Data_block_1".data_baru2[51] := "Suhu_Kiri";
   END_IF;
   IF #_w1 AND ("Data_block_1".counter_datasuhu = 53) THEN
       "Data_block_1".data_baru2[52] := "Suhu_Kiri";
   END_IF;
   IF #_w1 AND ("Data_block_1".counter_datasuhu = 54) THEN
       "Data_block_1".data_baru2[53] := "Suhu_Kiri";
   END_IF;
   IF #_w1 AND ("Data_block_1".counter_datasuhu = 55) THEN
       "Data_block_1".data_baru2[54] := "Suhu_Kiri";
   END_IF;
   IF #_w1 AND ("Data_block_1".counter_datasuhu = 56) THEN
       "Data_block_1".data_baru2[55] := "Suhu_Kiri";
   END_IF;
   IF #_w1 AND ("Data_block_1".counter_datasuhu = 57) THEN
       "Data_block_1".data_baru2[56] := "Suhu_Kiri";
   END_IF;
   IF #_w1 AND ("Data_block_1".counter_datasuhu = 58) THEN
       "Data_block_1".data_baru2[57] := "Suhu_Kiri";
   END_IF;
   IF #_w1 AND ("Data_block_1".counter_datasuhu = 59) THEN
       "Data_block_1".data_baru2[58] := "Suhu_Kiri";
   END_IF;
   IF #_w1 AND ("Data_block_1".counter_datasuhu = 60) THEN
       "Data_block_1".data_baru2[59] := "Suhu_Kiri";
   END_IF;
   IF #_w1 AND ("Data_block_1".counter_datasuhu = 61) THEN
       "Data_block_1".data_baru2[60] := "Suhu_Kiri";
   END_IF;
   IF #_w1 AND ("Data_block_1".counter_datasuhu = 62) THEN
       "Data_block_1".data_baru2[61] := "Suhu_Kiri";
   END_IF;
   IF #_w1 AND ("Data_block_1".counter_datasuhu = 63) THEN
       "Data_block_1".data_baru2[62] := "Suhu_Kiri";
   END_IF;
   IF #_w1 AND ("Data_block_1".counter_datasuhu = 64) THEN
       "Data_block_1".data_baru2[63] := "Suhu_Kiri";
   END_IF;
   IF #_w1 AND ("Data_block_1".counter_datasuhu = 65) THEN
       "Data_block_1".data_baru2[64] := "Suhu_Kiri";
   END_IF;
   IF #_w1 AND ("Data_block_1".counter_datasuhu = 66) THEN
       "Data_block_1".data_baru2[65] := "Suhu_Kiri";
   END_IF;
   IF #_w1 AND ("Data_block_1".counter_datasuhu = 67) THEN
       "Data_block_1".data_baru2[66] := "Suhu_Kiri";
   END_IF;
   IF #_w1 AND ("Data_block_1".counter_datasuhu = 68) THEN
       "Data_block_1".data_baru2[67] := "Suhu_Kiri";
   END_IF;
   IF #_w1 AND ("Data_block_1".counter_datasuhu = 69) THEN
       "Data_block_1".data_baru2[68] := "Suhu_Kiri";
   END_IF;
   IF #_w1 AND ("Data_block_1".counter_datasuhu = 70) THEN
       "Data_block_1".data_baru2[69] := "Suhu_Kiri";
   END_IF;
   IF #_w1 AND ("Data_block_1".counter_datasuhu = 71) THEN
       "Data_block_1".data_baru2[70] := "Suhu_Kiri";
   END_IF;
   IF #_w1 AND ("Data_block_1".counter_datasuhu = 72) THEN
       "Data_block_1".data_baru2[71] := "Suhu_Kiri";
   END_IF;
   IF #_w1 AND ("Data_block_1".counter_datasuhu = 73) THEN
       "Data_block_1".data_baru2[72] := "Suhu_Kiri";
   END_IF;
   IF #_w1 AND ("Data_block_1".counter_datasuhu = 74) THEN
       "Data_block_1".data_baru2[73] := "Suhu_Kiri";
   END_IF;
   IF #_w1 AND ("Data_block_1".counter_datasuhu = 75) THEN
       "Data_block_1".data_baru2[74] := "Suhu_Kiri";
   END_IF;
   IF #_w1 AND ("Data_block_1".counter_datasuhu = 76) THEN
       "Data_block_1".data_baru2[75] := "Suhu_Kiri";
   END_IF;
   IF #_w1 AND ("Data_block_1".counter_datasuhu = 77) THEN
       "Data_block_1".data_baru2[76] := "Suhu_Kiri";
   END_IF;
   IF #_w1 AND ("Data_block_1".counter_datasuhu = 78) THEN
       "Data_block_1".data_baru2[77] := "Suhu_Kiri";
   END_IF;
   IF #_w1 AND ("Data_block_1".counter_datasuhu = 79) THEN
       "Data_block_1".data_baru2[78] := "Suhu_Kiri";
   END_IF;
   IF #_w1 AND ("Data_block_1".counter_datasuhu = 80) THEN
       "Data_block_1".data_baru2[79] := "Suhu_Kiri";
   END_IF;
   IF #_w1 AND ("Data_block_1".counter_datasuhu = 81) THEN
       "Data_block_1".data_baru2[80] := "Suhu_Kiri";
   END_IF;
   IF #_w1 AND ("Data_block_1".counter_datasuhu = 82) THEN
       "Data_block_1".data_baru2[81] := "Suhu_Kiri";
   END_IF;
   IF #_w1 AND ("Data_block_1".counter_datasuhu = 83) THEN
       "Data_block_1".data_baru2[82] := "Suhu_Kiri";
   END_IF;
   IF #_w1 AND ("Data_block_1".counter_datasuhu = 84) THEN
       "Data_block_1".data_baru2[83] := "Suhu_Kiri";
   END_IF;
   IF #_w1 AND ("Data_block_1".counter_datasuhu = 85) THEN
       "Data_block_1".data_baru2[84] := "Suhu_Kiri";
   END_IF;
   IF #_w1 AND ("Data_block_1".counter_datasuhu = 86) THEN
       "Data_block_1".data_baru2[85] := "Suhu_Kiri";
   END_IF;
   IF #_w1 AND ("Data_block_1".counter_datasuhu = 87) THEN
       "Data_block_1".data_baru2[86] := "Suhu_Kiri";
   END_IF;
   IF #_w1 AND ("Data_block_1".counter_datasuhu = 88) THEN
       "Data_block_1".data_baru2[87] := "Suhu_Kiri";
   END_IF;
   IF #_w1 AND ("Data_block_1".counter_datasuhu = 89) THEN
       "Data_block_1".data_baru2[88] := "Suhu_Kiri";
   END_IF;
   IF #_w1 AND ("Data_block_1".counter_datasuhu = 90) THEN
       "Data_block_1".data_baru2[89] := "Suhu_Kiri";
   END_IF;
   IF #_w1 AND ("Data_block_1".counter_datasuhu = 91) THEN
       "Data_block_1".data_baru2[90] := "Suhu_Kiri";
   END_IF;
   IF #_w1 AND ("Data_block_1".counter_datasuhu = 92) THEN
       "Data_block_1".data_baru2[91] := "Suhu_Kiri";
   END_IF;
   IF #_w1 AND ("Data_block_1".counter_datasuhu = 93) THEN
       "Data_block_1".data_baru2[92] := "Suhu_Kiri";
   END_IF;
   IF #_w1 AND ("Data_block_1".counter_datasuhu = 94) THEN
       "Data_block_1".data_baru2[93] := "Suhu_Kiri";
   END_IF;
   IF #_w1 AND ("Data_block_1".counter_datasuhu = 95) THEN
       "Data_block_1".data_baru2[94] := "Suhu_Kiri";
   END_IF;
   IF #_w1 AND ("Data_block_1".counter_datasuhu = 96) THEN
       "Data_block_1".data_baru2[95] := "Suhu_Kiri";
   END_IF;
   IF #_w1 AND ("Data_block_1".counter_datasuhu = 97) THEN
       "Data_block_1".data_baru2[96] := "Suhu_Kiri";
   END_IF;
   IF #_w1 AND ("Data_block_1".counter_datasuhu = 98) THEN
       "Data_block_1".data_baru2[97] := "Suhu_Kiri";
   END_IF;
   IF #_w1 AND ("Data_block_1".counter_datasuhu = 99) THEN
       "Data_block_1".data_baru2[98] := "Suhu_Kiri";
   END_IF;
   IF #_w1 AND ("Data_block_1".counter_datasuhu = 100) THEN
       "Data_block_1".data_baru2[99] := "Suhu_Kiri";
   END_IF;
END_REGION

REGION Network 25: counter (roda)
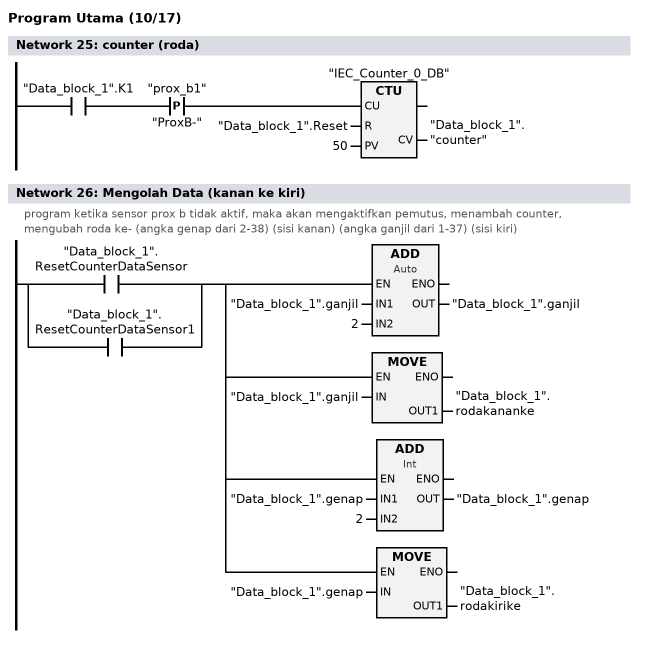
   #_w1 := "Data_block_1".K1 AND "prox_b1" AND NOT "ProxB-";   // rising edge of "prox_b1"
   "ProxB-" := "prox_b1";
   "IEC_Counter_0_DB".CTU(CU := #_w1, R := "Data_block_1".Reset, PV := 50, CV => "Data_block_1"."counter");
END_REGION

REGION Network 26: Mengolah Data (kanan ke kiri)
   // program ketika sensor prox b tidak aktif, maka akan mengaktifkan pemutus, menambah counter, mengubah roda ke- (angka genap dari 2-38) (sisi kanan) (angka ganjil dari 1-37) (sisi kiri)
   RUNG wire#powerrail
      Contact( "Data_block_1".ResetCounterDataSensor )
      wire#w1
      Add(in1 := "Data_block_1".ganjil, in2 := 2, out => "Data_block_1".ganjil)
   END_RUNG
   RUNG wire#powerrail
      Contact( "Data_block_1".ResetCounterDataSensor1 )
   END_RUNG wire#w1
   RUNG wire#w1
      Move(in := "Data_block_1".ganjil, out1 => "Data_block_1".rodakananke)
   END_RUNG
   RUNG wire#w1
      { S7_Templates := "SrcType := Int" } Add(in1 := "Data_block_1".genap, in2 := 2, out => "Data_block_1".genap)
   END_RUNG
   RUNG wire#w1
      Move(in := "Data_block_1".genap, out1 => "Data_block_1".rodakirike)
   END_RUNG
   // the same network as SCL:
   IF "Data_block_1".ResetCounterDataSensor OR "Data_block_1".ResetCounterDataSensor1 THEN
       "Data_block_1".ganjil := "Data_block_1".ganjil + 2;
       "Data_block_1".rodakananke := "Data_block_1".ganjil;
       "Data_block_1".genap := "Data_block_1".genap + 2;
       "Data_block_1".rodakirike := "Data_block_1".genap;
   END_IF;
END_REGION

REGION Network 27: Menentukan Nilai Tengah (kanan ke kiri)
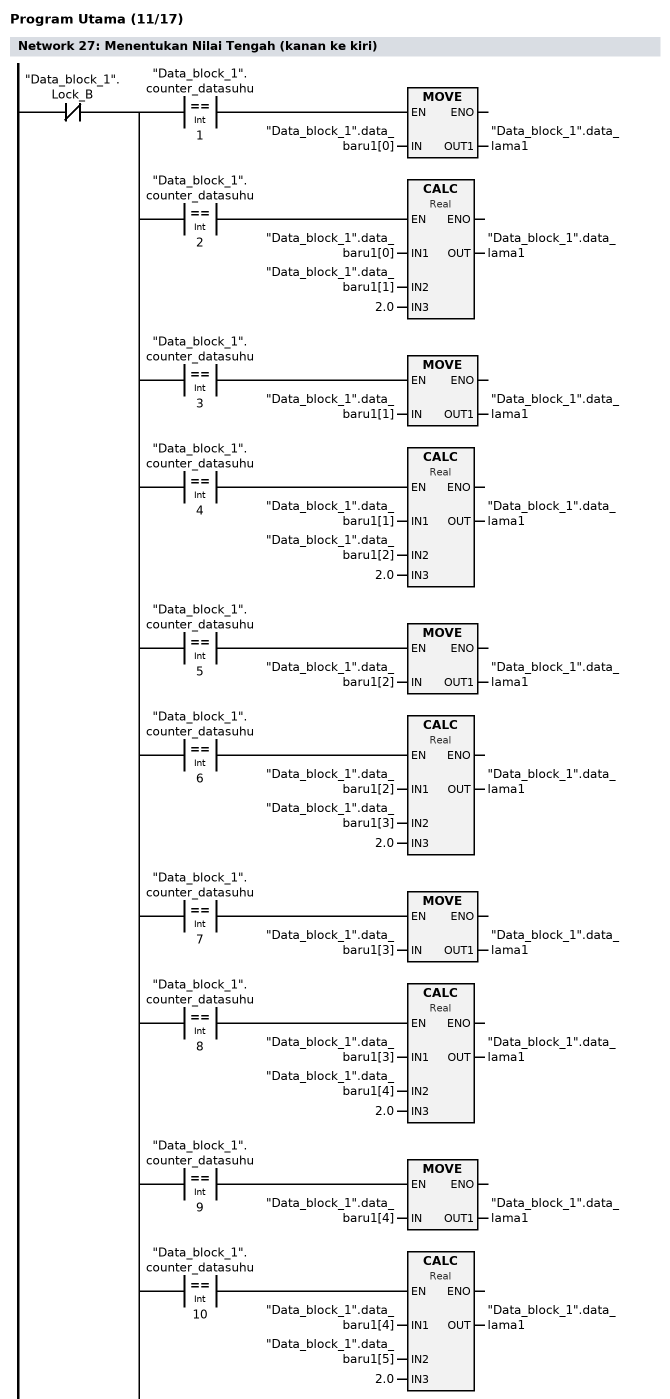
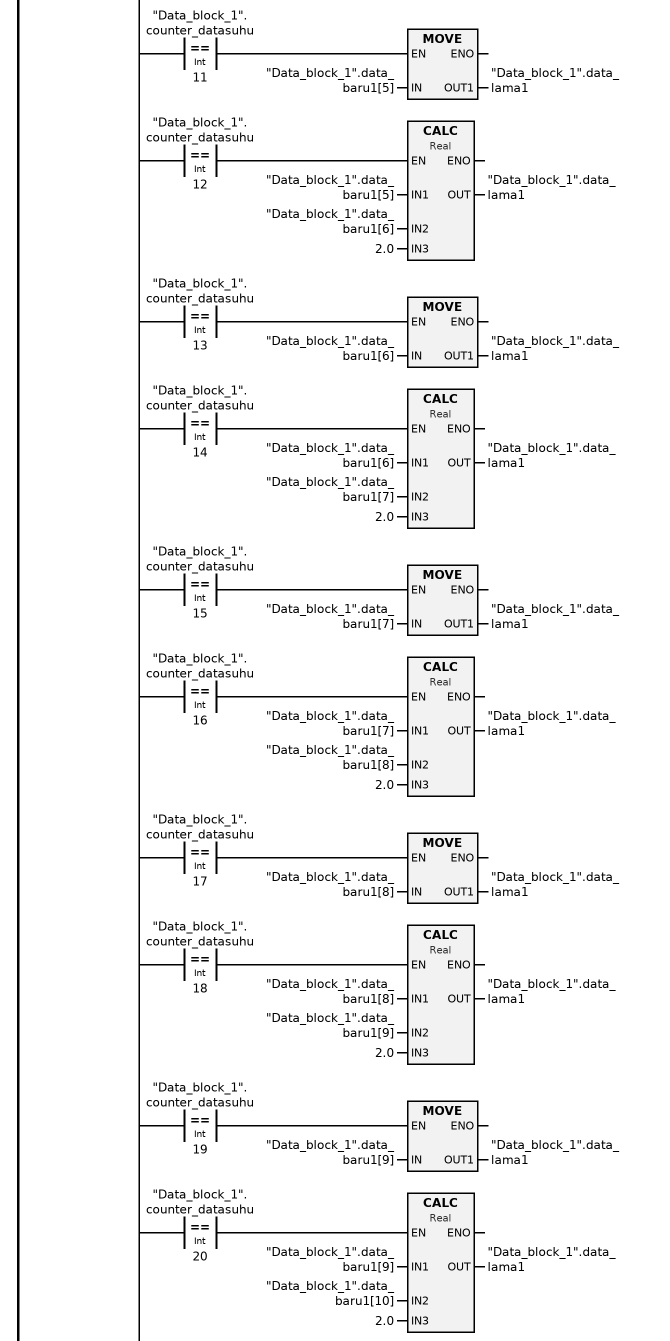
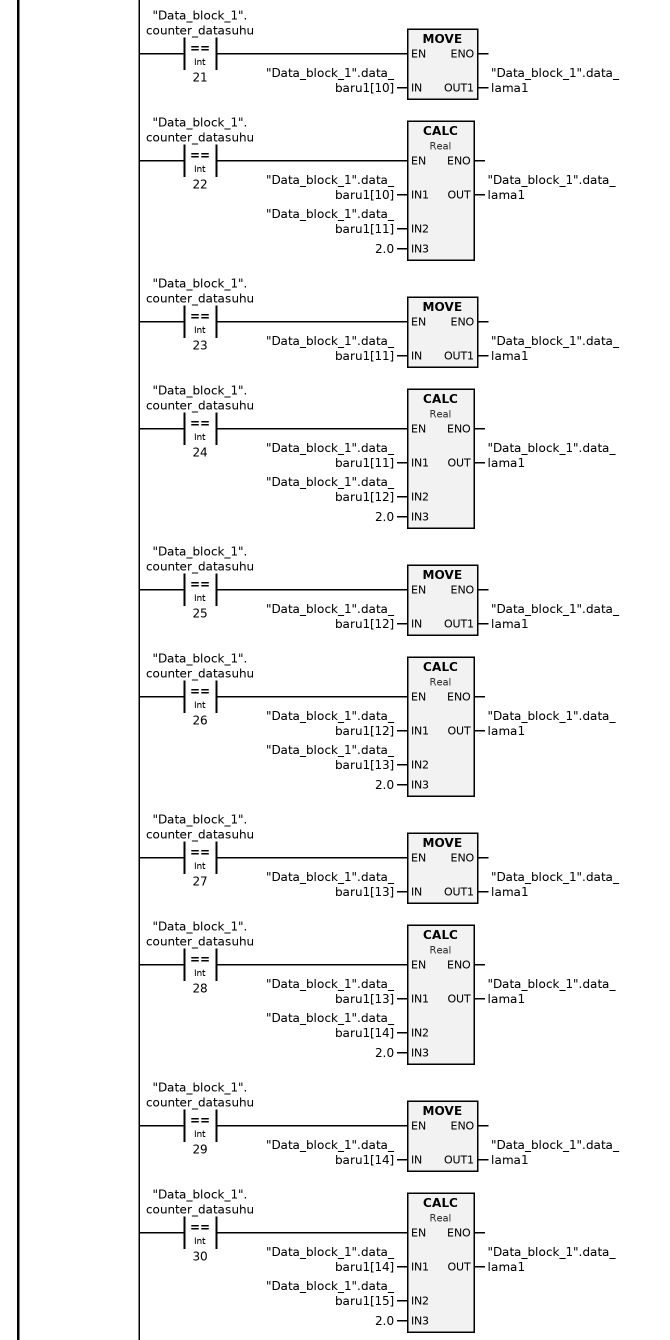
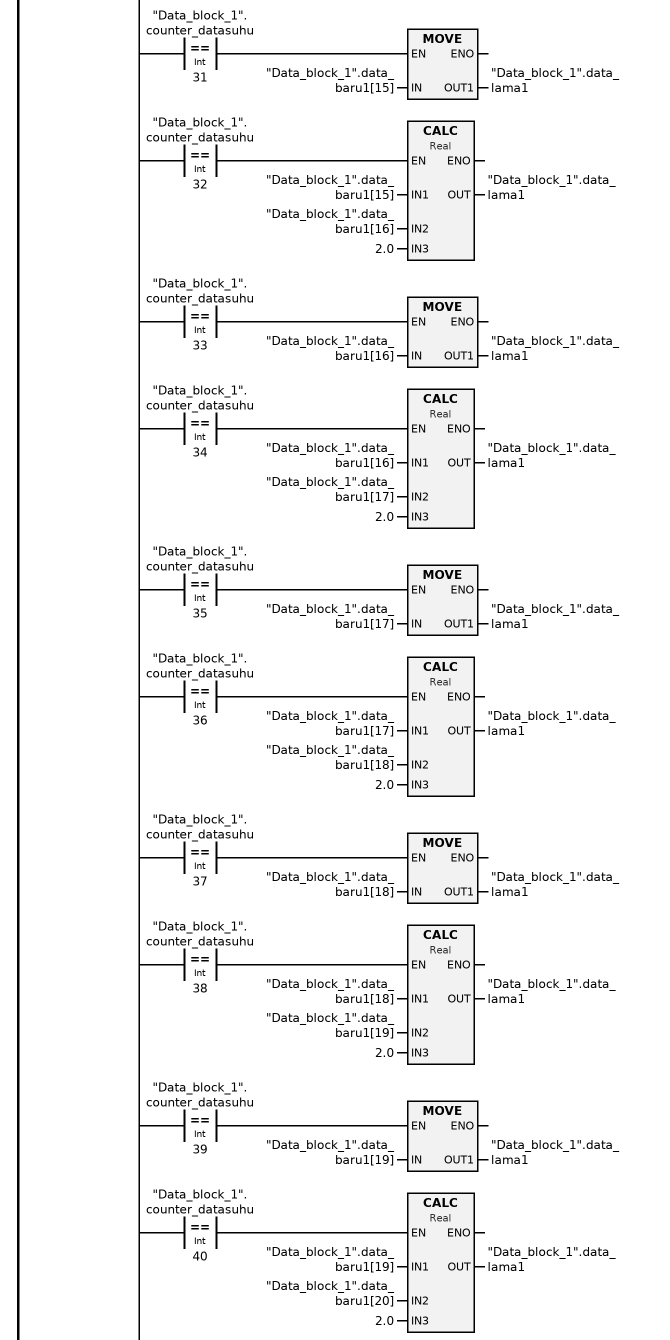
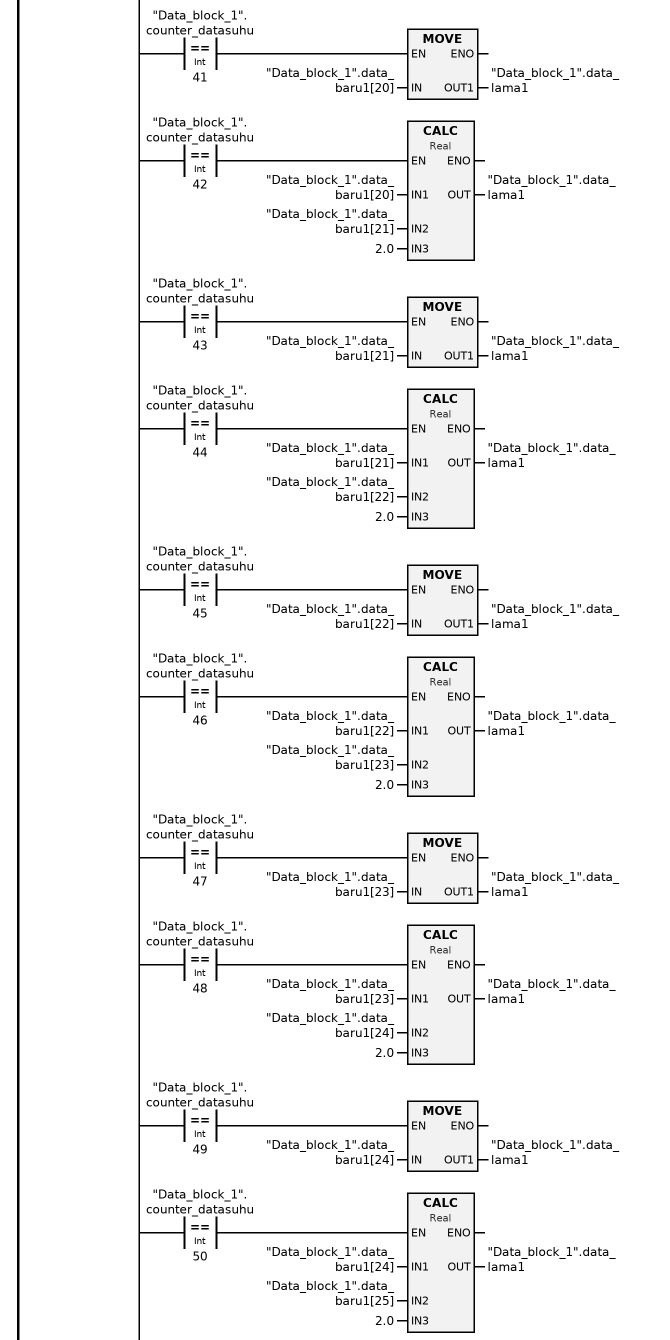
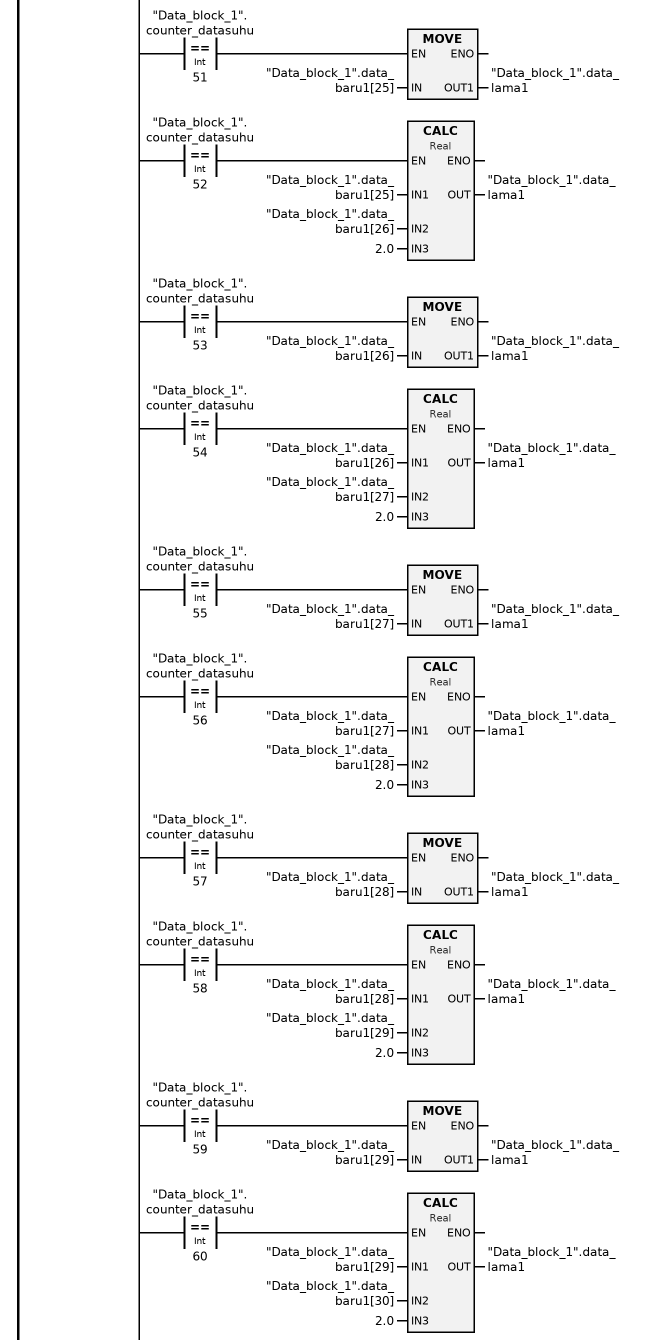
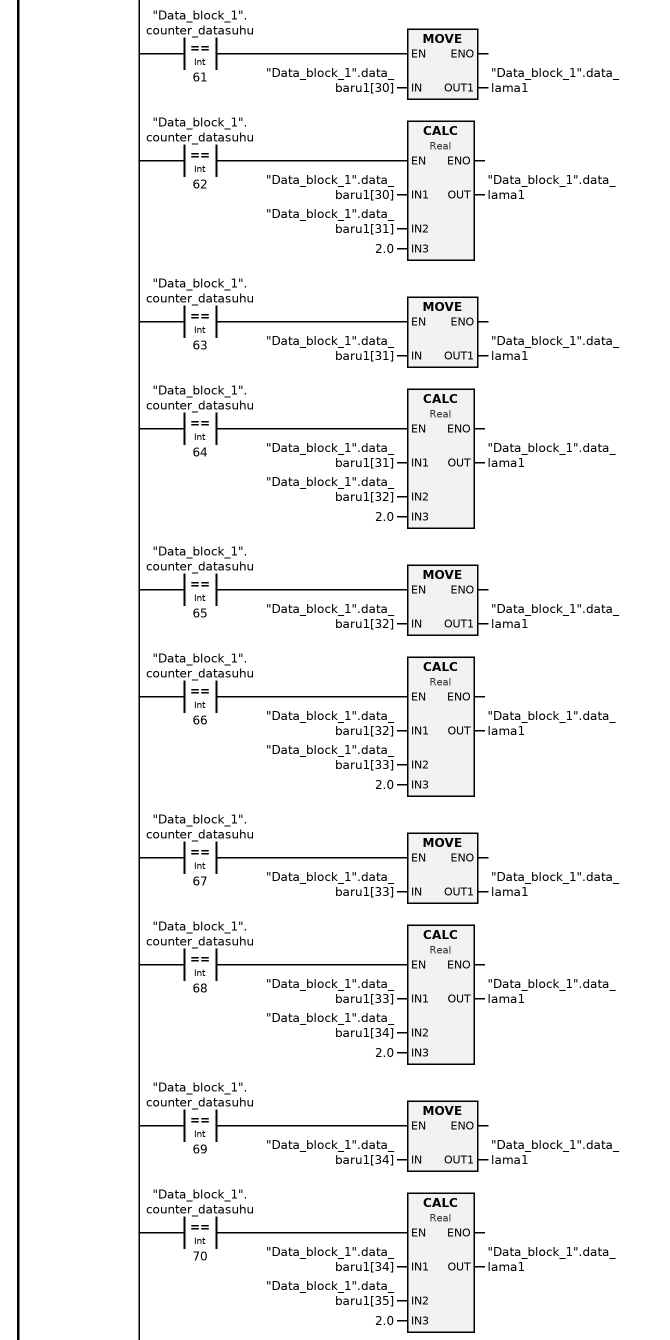
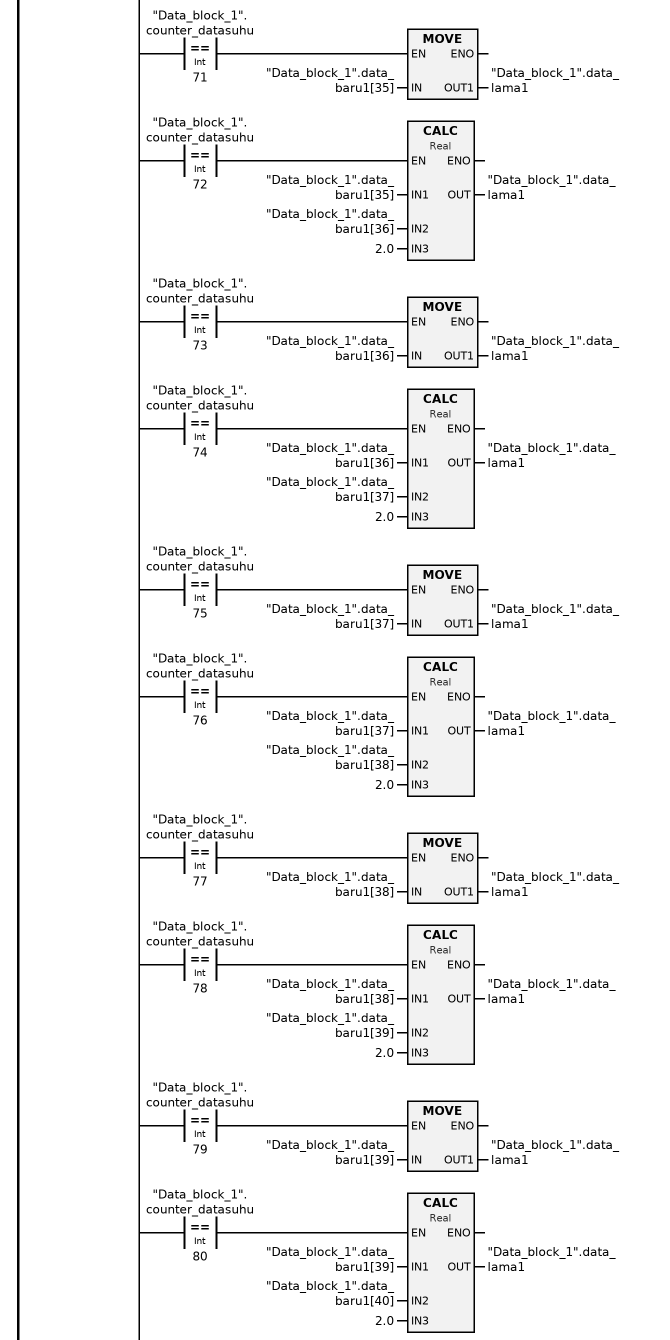
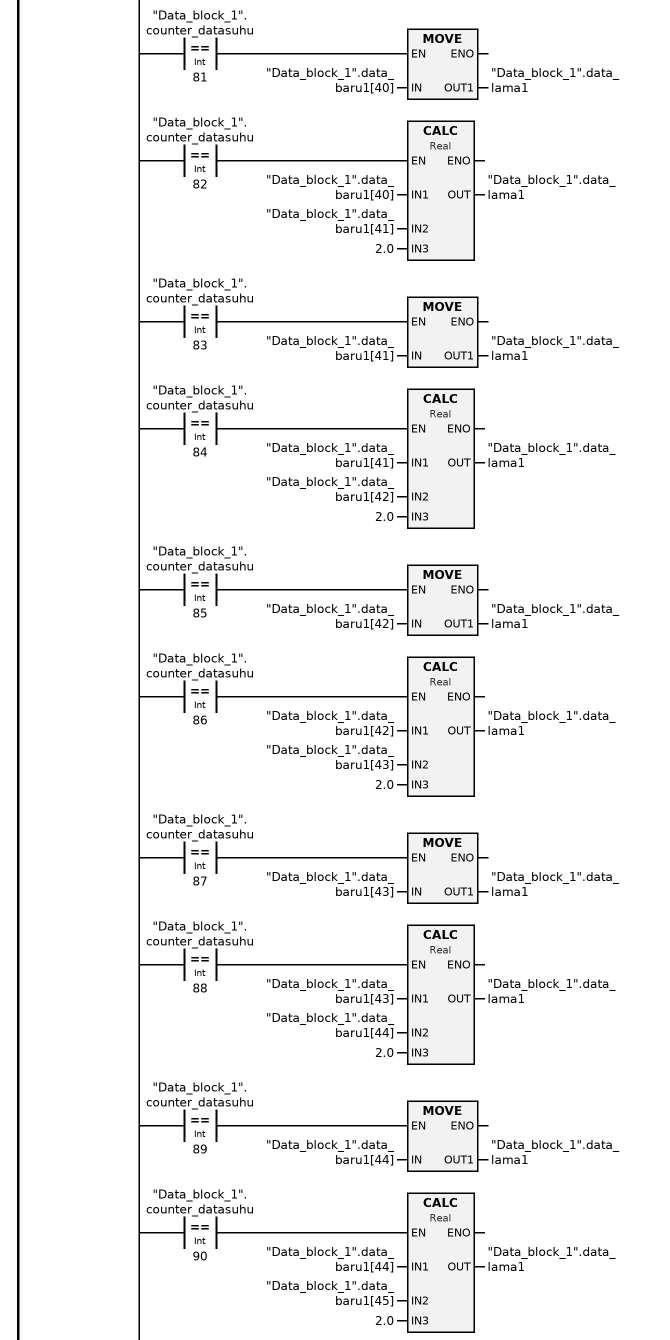
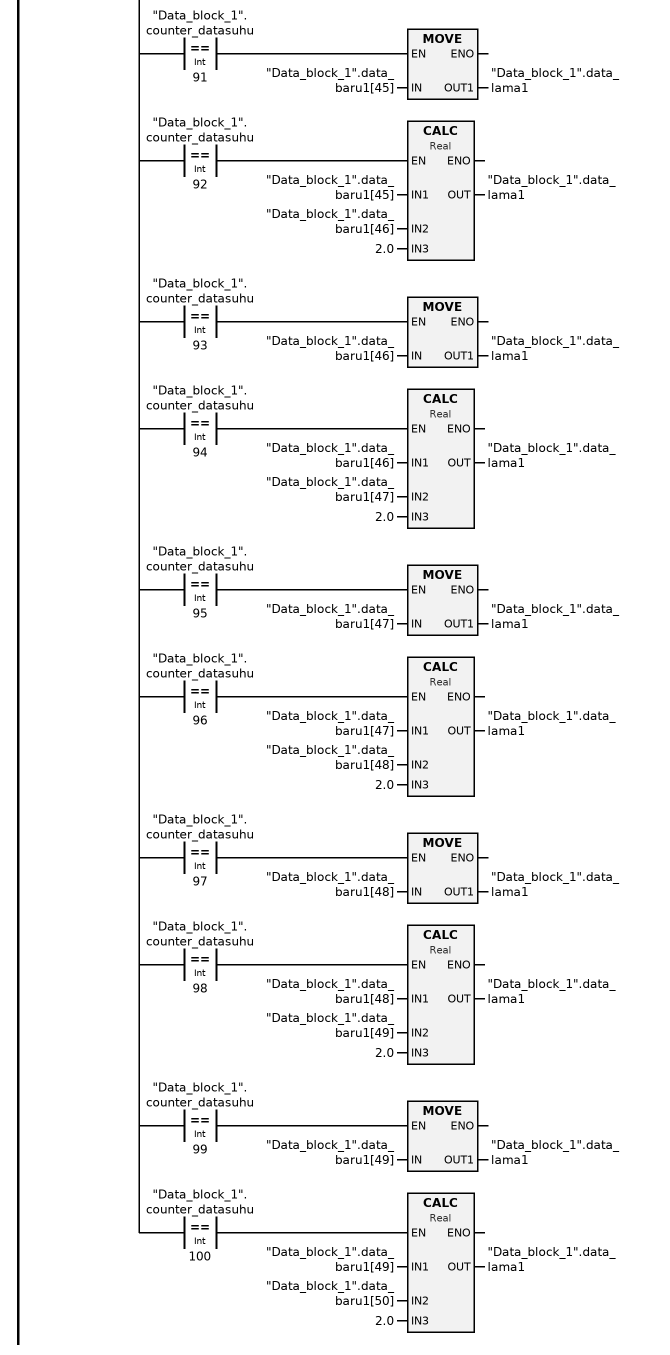
   #_w1 := NOT "Data_block_1".Lock_B;
   IF #_w1 AND ("Data_block_1".counter_datasuhu = 1) THEN
       "Data_block_1".data_lama1 := "Data_block_1".data_baru1[0];
   END_IF;
   IF #_w1 AND ("Data_block_1".counter_datasuhu = 2) THEN
       CALC(in1 := "Data_block_1".data_baru1[0],
            in2 := "Data_block_1".data_baru1[1],
            in3 := 2.0,
            out => "Data_block_1".data_lama1);
   END_IF;
   IF #_w1 AND ("Data_block_1".counter_datasuhu = 3) THEN
       "Data_block_1".data_lama1 := "Data_block_1".data_baru1[1];
   END_IF;
   IF #_w1 AND ("Data_block_1".counter_datasuhu = 4) THEN
       CALC(in1 := "Data_block_1".data_baru1[1],
            in2 := "Data_block_1".data_baru1[2],
            in3 := 2.0,
            out => "Data_block_1".data_lama1);
   END_IF;
   IF #_w1 AND ("Data_block_1".counter_datasuhu = 5) THEN
       "Data_block_1".data_lama1 := "Data_block_1".data_baru1[2];
   END_IF;
   IF #_w1 AND ("Data_block_1".counter_datasuhu = 6) THEN
       CALC(in1 := "Data_block_1".data_baru1[2],
            in2 := "Data_block_1".data_baru1[3],
            in3 := 2.0,
            out => "Data_block_1".data_lama1);
   END_IF;
   IF #_w1 AND ("Data_block_1".counter_datasuhu = 7) THEN
       "Data_block_1".data_lama1 := "Data_block_1".data_baru1[3];
   END_IF;
   IF #_w1 AND ("Data_block_1".counter_datasuhu = 8) THEN
       CALC(in1 := "Data_block_1".data_baru1[3],
            in2 := "Data_block_1".data_baru1[4],
            in3 := 2.0,
            out => "Data_block_1".data_lama1);
   END_IF;
   IF #_w1 AND ("Data_block_1".counter_datasuhu = 9) THEN
       "Data_block_1".data_lama1 := "Data_block_1".data_baru1[4];
   END_IF;
   IF #_w1 AND ("Data_block_1".counter_datasuhu = 10) THEN
       CALC(in1 := "Data_block_1".data_baru1[4],
            in2 := "Data_block_1".data_baru1[5],
            in3 := 2.0,
            out => "Data_block_1".data_lama1);
   END_IF;
   IF #_w1 AND ("Data_block_1".counter_datasuhu = 11) THEN
       "Data_block_1".data_lama1 := "Data_block_1".data_baru1[5];
   END_IF;
   IF #_w1 AND ("Data_block_1".counter_datasuhu = 12) THEN
       CALC(in1 := "Data_block_1".data_baru1[5],
            in2 := "Data_block_1".data_baru1[6],
            in3 := 2.0,
            out => "Data_block_1".data_lama1);
   END_IF;
   IF #_w1 AND ("Data_block_1".counter_datasuhu = 13) THEN
       "Data_block_1".data_lama1 := "Data_block_1".data_baru1[6];
   END_IF;
   IF #_w1 AND ("Data_block_1".counter_datasuhu = 14) THEN
       CALC(in1 := "Data_block_1".data_baru1[6],
            in2 := "Data_block_1".data_baru1[7],
            in3 := 2.0,
            out => "Data_block_1".data_lama1);
   END_IF;
   IF #_w1 AND ("Data_block_1".counter_datasuhu = 15) THEN
       "Data_block_1".data_lama1 := "Data_block_1".data_baru1[7];
   END_IF;
   IF #_w1 AND ("Data_block_1".counter_datasuhu = 16) THEN
       CALC(in1 := "Data_block_1".data_baru1[7],
            in2 := "Data_block_1".data_baru1[8],
            in3 := 2.0,
            out => "Data_block_1".data_lama1);
   END_IF;
   IF #_w1 AND ("Data_block_1".counter_datasuhu = 17) THEN
       "Data_block_1".data_lama1 := "Data_block_1".data_baru1[8];
   END_IF;
   IF #_w1 AND ("Data_block_1".counter_datasuhu = 18) THEN
       CALC(in1 := "Data_block_1".data_baru1[8],
            in2 := "Data_block_1".data_baru1[9],
            in3 := 2.0,
            out => "Data_block_1".data_lama1);
   END_IF;
   IF #_w1 AND ("Data_block_1".counter_datasuhu = 19) THEN
       "Data_block_1".data_lama1 := "Data_block_1".data_baru1[9];
   END_IF;
   IF #_w1 AND ("Data_block_1".counter_datasuhu = 20) THEN
       CALC(in1 := "Data_block_1".data_baru1[9],
            in2 := "Data_block_1".data_baru1[10],
            in3 := 2.0,
            out => "Data_block_1".data_lama1);
   END_IF;
   IF #_w1 AND ("Data_block_1".counter_datasuhu = 21) THEN
       "Data_block_1".data_lama1 := "Data_block_1".data_baru1[10];
   END_IF;
   IF #_w1 AND ("Data_block_1".counter_datasuhu = 22) THEN
       CALC(in1 := "Data_block_1".data_baru1[10],
            in2 := "Data_block_1".data_baru1[11],
            in3 := 2.0,
            out => "Data_block_1".data_lama1);
   END_IF;
   IF #_w1 AND ("Data_block_1".counter_datasuhu = 23) THEN
       "Data_block_1".data_lama1 := "Data_block_1".data_baru1[11];
   END_IF;
   IF #_w1 AND ("Data_block_1".counter_datasuhu = 24) THEN
       CALC(in1 := "Data_block_1".data_baru1[11],
            in2 := "Data_block_1".data_baru1[12],
            in3 := 2.0,
            out => "Data_block_1".data_lama1);
   END_IF;
   IF #_w1 AND ("Data_block_1".counter_datasuhu = 25) THEN
       "Data_block_1".data_lama1 := "Data_block_1".data_baru1[12];
   END_IF;
   IF #_w1 AND ("Data_block_1".counter_datasuhu = 26) THEN
       CALC(in1 := "Data_block_1".data_baru1[12],
            in2 := "Data_block_1".data_baru1[13],
            in3 := 2.0,
            out => "Data_block_1".data_lama1);
   END_IF;
   IF #_w1 AND ("Data_block_1".counter_datasuhu = 27) THEN
       "Data_block_1".data_lama1 := "Data_block_1".data_baru1[13];
   END_IF;
   IF #_w1 AND ("Data_block_1".counter_datasuhu = 28) THEN
       CALC(in1 := "Data_block_1".data_baru1[13],
            in2 := "Data_block_1".data_baru1[14],
            in3 := 2.0,
            out => "Data_block_1".data_lama1);
   END_IF;
   IF #_w1 AND ("Data_block_1".counter_datasuhu = 29) THEN
       "Data_block_1".data_lama1 := "Data_block_1".data_baru1[14];
   END_IF;
   IF #_w1 AND ("Data_block_1".counter_datasuhu = 30) THEN
       CALC(in1 := "Data_block_1".data_baru1[14],
            in2 := "Data_block_1".data_baru1[15],
            in3 := 2.0,
            out => "Data_block_1".data_lama1);
   END_IF;
   IF #_w1 AND ("Data_block_1".counter_datasuhu = 31) THEN
       "Data_block_1".data_lama1 := "Data_block_1".data_baru1[15];
   END_IF;
   IF #_w1 AND ("Data_block_1".counter_datasuhu = 32) THEN
       CALC(in1 := "Data_block_1".data_baru1[15],
            in2 := "Data_block_1".data_baru1[16],
            in3 := 2.0,
            out => "Data_block_1".data_lama1);
   END_IF;
   IF #_w1 AND ("Data_block_1".counter_datasuhu = 33) THEN
       "Data_block_1".data_lama1 := "Data_block_1".data_baru1[16];
   END_IF;
   IF #_w1 AND ("Data_block_1".counter_datasuhu = 34) THEN
       CALC(in1 := "Data_block_1".data_baru1[16],
            in2 := "Data_block_1".data_baru1[17],
            in3 := 2.0,
            out => "Data_block_1".data_lama1);
   END_IF;
   IF #_w1 AND ("Data_block_1".counter_datasuhu = 35) THEN
       "Data_block_1".data_lama1 := "Data_block_1".data_baru1[17];
   END_IF;
   IF #_w1 AND ("Data_block_1".counter_datasuhu = 36) THEN
       CALC(in1 := "Data_block_1".data_baru1[17],
            in2 := "Data_block_1".data_baru1[18],
            in3 := 2.0,
            out => "Data_block_1".data_lama1);
   END_IF;
   IF #_w1 AND ("Data_block_1".counter_datasuhu = 37) THEN
       "Data_block_1".data_lama1 := "Data_block_1".data_baru1[18];
   END_IF;
   IF #_w1 AND ("Data_block_1".counter_datasuhu = 38) THEN
       CALC(in1 := "Data_block_1".data_baru1[18],
            in2 := "Data_block_1".data_baru1[19],
            in3 := 2.0,
            out => "Data_block_1".data_lama1);
   END_IF;
   IF #_w1 AND ("Data_block_1".counter_datasuhu = 39) THEN
       "Data_block_1".data_lama1 := "Data_block_1".data_baru1[19];
   END_IF;
   IF #_w1 AND ("Data_block_1".counter_datasuhu = 40) THEN
       CALC(in1 := "Data_block_1".data_baru1[19],
            in2 := "Data_block_1".data_baru1[20],
            in3 := 2.0,
            out => "Data_block_1".data_lama1);
   END_IF;
   IF #_w1 AND ("Data_block_1".counter_datasuhu = 41) THEN
       "Data_block_1".data_lama1 := "Data_block_1".data_baru1[20];
   END_IF;
   IF #_w1 AND ("Data_block_1".counter_datasuhu = 42) THEN
       CALC(in1 := "Data_block_1".data_baru1[20],
            in2 := "Data_block_1".data_baru1[21],
            in3 := 2.0,
            out => "Data_block_1".data_lama1);
   END_IF;
   IF #_w1 AND ("Data_block_1".counter_datasuhu = 43) THEN
       "Data_block_1".data_lama1 := "Data_block_1".data_baru1[21];
   END_IF;
   IF #_w1 AND ("Data_block_1".counter_datasuhu = 44) THEN
       CALC(in1 := "Data_block_1".data_baru1[21],
            in2 := "Data_block_1".data_baru1[22],
            in3 := 2.0,
            out => "Data_block_1".data_lama1);
   END_IF;
   IF #_w1 AND ("Data_block_1".counter_datasuhu = 45) THEN
       "Data_block_1".data_lama1 := "Data_block_1".data_baru1[22];
   END_IF;
   IF #_w1 AND ("Data_block_1".counter_datasuhu = 46) THEN
       CALC(in1 := "Data_block_1".data_baru1[22],
            in2 := "Data_block_1".data_baru1[23],
            in3 := 2.0,
            out => "Data_block_1".data_lama1);
   END_IF;
   IF #_w1 AND ("Data_block_1".counter_datasuhu = 47) THEN
       "Data_block_1".data_lama1 := "Data_block_1".data_baru1[23];
   END_IF;
   IF #_w1 AND ("Data_block_1".counter_datasuhu = 48) THEN
       CALC(in1 := "Data_block_1".data_baru1[23],
            in2 := "Data_block_1".data_baru1[24],
            in3 := 2.0,
            out => "Data_block_1".data_lama1);
   END_IF;
   IF #_w1 AND ("Data_block_1".counter_datasuhu = 49) THEN
       "Data_block_1".data_lama1 := "Data_block_1".data_baru1[24];
   END_IF;
   IF #_w1 AND ("Data_block_1".counter_datasuhu = 50) THEN
       CALC(in1 := "Data_block_1".data_baru1[24],
            in2 := "Data_block_1".data_baru1[25],
            in3 := 2.0,
            out => "Data_block_1".data_lama1);
   END_IF;
   IF #_w1 AND ("Data_block_1".counter_datasuhu = 51) THEN
       "Data_block_1".data_lama1 := "Data_block_1".data_baru1[25];
   END_IF;
   IF #_w1 AND ("Data_block_1".counter_datasuhu = 52) THEN
       CALC(in1 := "Data_block_1".data_baru1[25],
            in2 := "Data_block_1".data_baru1[26],
            in3 := 2.0,
            out => "Data_block_1".data_lama1);
   END_IF;
   IF #_w1 AND ("Data_block_1".counter_datasuhu = 53) THEN
       "Data_block_1".data_lama1 := "Data_block_1".data_baru1[26];
   END_IF;
   IF #_w1 AND ("Data_block_1".counter_datasuhu = 54) THEN
       CALC(in1 := "Data_block_1".data_baru1[26],
            in2 := "Data_block_1".data_baru1[27],
            in3 := 2.0,
            out => "Data_block_1".data_lama1);
   END_IF;
   IF #_w1 AND ("Data_block_1".counter_datasuhu = 55) THEN
       "Data_block_1".data_lama1 := "Data_block_1".data_baru1[27];
   END_IF;
   IF #_w1 AND ("Data_block_1".counter_datasuhu = 56) THEN
       CALC(in1 := "Data_block_1".data_baru1[27],
            in2 := "Data_block_1".data_baru1[28],
            in3 := 2.0,
            out => "Data_block_1".data_lama1);
   END_IF;
   IF #_w1 AND ("Data_block_1".counter_datasuhu = 57) THEN
       "Data_block_1".data_lama1 := "Data_block_1".data_baru1[28];
   END_IF;
   IF #_w1 AND ("Data_block_1".counter_datasuhu = 58) THEN
       CALC(in1 := "Data_block_1".data_baru1[28],
            in2 := "Data_block_1".data_baru1[29],
            in3 := 2.0,
            out => "Data_block_1".data_lama1);
   END_IF;
   IF #_w1 AND ("Data_block_1".counter_datasuhu = 59) THEN
       "Data_block_1".data_lama1 := "Data_block_1".data_baru1[29];
   END_IF;
   IF #_w1 AND ("Data_block_1".counter_datasuhu = 60) THEN
       CALC(in1 := "Data_block_1".data_baru1[29],
            in2 := "Data_block_1".data_baru1[30],
            in3 := 2.0,
            out => "Data_block_1".data_lama1);
   END_IF;
   IF #_w1 AND ("Data_block_1".counter_datasuhu = 61) THEN
       "Data_block_1".data_lama1 := "Data_block_1".data_baru1[30];
   END_IF;
   IF #_w1 AND ("Data_block_1".counter_datasuhu = 62) THEN
       CALC(in1 := "Data_block_1".data_baru1[30],
            in2 := "Data_block_1".data_baru1[31],
            in3 := 2.0,
            out => "Data_block_1".data_lama1);
   END_IF;
   IF #_w1 AND ("Data_block_1".counter_datasuhu = 63) THEN
       "Data_block_1".data_lama1 := "Data_block_1".data_baru1[31];
   END_IF;
   IF #_w1 AND ("Data_block_1".counter_datasuhu = 64) THEN
       CALC(in1 := "Data_block_1".data_baru1[31],
            in2 := "Data_block_1".data_baru1[32],
            in3 := 2.0,
            out => "Data_block_1".data_lama1);
   END_IF;
   IF #_w1 AND ("Data_block_1".counter_datasuhu = 65) THEN
       "Data_block_1".data_lama1 := "Data_block_1".data_baru1[32];
   END_IF;
   IF #_w1 AND ("Data_block_1".counter_datasuhu = 66) THEN
       CALC(in1 := "Data_block_1".data_baru1[32],
            in2 := "Data_block_1".data_baru1[33],
            in3 := 2.0,
            out => "Data_block_1".data_lama1);
   END_IF;
   IF #_w1 AND ("Data_block_1".counter_datasuhu = 67) THEN
       "Data_block_1".data_lama1 := "Data_block_1".data_baru1[33];
   END_IF;
   IF #_w1 AND ("Data_block_1".counter_datasuhu = 68) THEN
       CALC(in1 := "Data_block_1".data_baru1[33],
            in2 := "Data_block_1".data_baru1[34],
            in3 := 2.0,
            out => "Data_block_1".data_lama1);
   END_IF;
   IF #_w1 AND ("Data_block_1".counter_datasuhu = 69) THEN
       "Data_block_1".data_lama1 := "Data_block_1".data_baru1[34];
   END_IF;
   IF #_w1 AND ("Data_block_1".counter_datasuhu = 70) THEN
       CALC(in1 := "Data_block_1".data_baru1[34],
            in2 := "Data_block_1".data_baru1[35],
            in3 := 2.0,
            out => "Data_block_1".data_lama1);
   END_IF;
   IF #_w1 AND ("Data_block_1".counter_datasuhu = 71) THEN
       "Data_block_1".data_lama1 := "Data_block_1".data_baru1[35];
   END_IF;
   IF #_w1 AND ("Data_block_1".counter_datasuhu = 72) THEN
       CALC(in1 := "Data_block_1".data_baru1[35],
            in2 := "Data_block_1".data_baru1[36],
            in3 := 2.0,
            out => "Data_block_1".data_lama1);
   END_IF;
   IF #_w1 AND ("Data_block_1".counter_datasuhu = 73) THEN
       "Data_block_1".data_lama1 := "Data_block_1".data_baru1[36];
   END_IF;
   IF #_w1 AND ("Data_block_1".counter_datasuhu = 74) THEN
       CALC(in1 := "Data_block_1".data_baru1[36],
            in2 := "Data_block_1".data_baru1[37],
            in3 := 2.0,
            out => "Data_block_1".data_lama1);
   END_IF;
   IF #_w1 AND ("Data_block_1".counter_datasuhu = 75) THEN
       "Data_block_1".data_lama1 := "Data_block_1".data_baru1[37];
   END_IF;
   IF #_w1 AND ("Data_block_1".counter_datasuhu = 76) THEN
       CALC(in1 := "Data_block_1".data_baru1[37],
            in2 := "Data_block_1".data_baru1[38],
            in3 := 2.0,
            out => "Data_block_1".data_lama1);
   END_IF;
   IF #_w1 AND ("Data_block_1".counter_datasuhu = 77) THEN
       "Data_block_1".data_lama1 := "Data_block_1".data_baru1[38];
   END_IF;
   IF #_w1 AND ("Data_block_1".counter_datasuhu = 78) THEN
       CALC(in1 := "Data_block_1".data_baru1[38],
            in2 := "Data_block_1".data_baru1[39],
            in3 := 2.0,
            out => "Data_block_1".data_lama1);
   END_IF;
   IF #_w1 AND ("Data_block_1".counter_datasuhu = 79) THEN
       "Data_block_1".data_lama1 := "Data_block_1".data_baru1[39];
   END_IF;
   IF #_w1 AND ("Data_block_1".counter_datasuhu = 80) THEN
       CALC(in1 := "Data_block_1".data_baru1[39],
            in2 := "Data_block_1".data_baru1[40],
            in3 := 2.0,
            out => "Data_block_1".data_lama1);
   END_IF;
   IF #_w1 AND ("Data_block_1".counter_datasuhu = 81) THEN
       "Data_block_1".data_lama1 := "Data_block_1".data_baru1[40];
   END_IF;
   IF #_w1 AND ("Data_block_1".counter_datasuhu = 82) THEN
       CALC(in1 := "Data_block_1".data_baru1[40],
            in2 := "Data_block_1".data_baru1[41],
            in3 := 2.0,
            out => "Data_block_1".data_lama1);
   END_IF;
   IF #_w1 AND ("Data_block_1".counter_datasuhu = 83) THEN
       "Data_block_1".data_lama1 := "Data_block_1".data_baru1[41];
   END_IF;
   IF #_w1 AND ("Data_block_1".counter_datasuhu = 84) THEN
       CALC(in1 := "Data_block_1".data_baru1[41],
            in2 := "Data_block_1".data_baru1[42],
            in3 := 2.0,
            out => "Data_block_1".data_lama1);
   END_IF;
   IF #_w1 AND ("Data_block_1".counter_datasuhu = 85) THEN
       "Data_block_1".data_lama1 := "Data_block_1".data_baru1[42];
   END_IF;
   IF #_w1 AND ("Data_block_1".counter_datasuhu = 86) THEN
       CALC(in1 := "Data_block_1".data_baru1[42],
            in2 := "Data_block_1".data_baru1[43],
            in3 := 2.0,
            out => "Data_block_1".data_lama1);
   END_IF;
   IF #_w1 AND ("Data_block_1".counter_datasuhu = 87) THEN
       "Data_block_1".data_lama1 := "Data_block_1".data_baru1[43];
   END_IF;
   IF #_w1 AND ("Data_block_1".counter_datasuhu = 88) THEN
       CALC(in1 := "Data_block_1".data_baru1[43],
            in2 := "Data_block_1".data_baru1[44],
            in3 := 2.0,
            out => "Data_block_1".data_lama1);
   END_IF;
   IF #_w1 AND ("Data_block_1".counter_datasuhu = 89) THEN
       "Data_block_1".data_lama1 := "Data_block_1".data_baru1[44];
   END_IF;
   IF #_w1 AND ("Data_block_1".counter_datasuhu = 90) THEN
       CALC(in1 := "Data_block_1".data_baru1[44],
            in2 := "Data_block_1".data_baru1[45],
            in3 := 2.0,
            out => "Data_block_1".data_lama1);
   END_IF;
   IF #_w1 AND ("Data_block_1".counter_datasuhu = 91) THEN
       "Data_block_1".data_lama1 := "Data_block_1".data_baru1[45];
   END_IF;
   IF #_w1 AND ("Data_block_1".counter_datasuhu = 92) THEN
       CALC(in1 := "Data_block_1".data_baru1[45],
            in2 := "Data_block_1".data_baru1[46],
            in3 := 2.0,
            out => "Data_block_1".data_lama1);
   END_IF;
   IF #_w1 AND ("Data_block_1".counter_datasuhu = 93) THEN
       "Data_block_1".data_lama1 := "Data_block_1".data_baru1[46];
   END_IF;
   IF #_w1 AND ("Data_block_1".counter_datasuhu = 94) THEN
       CALC(in1 := "Data_block_1".data_baru1[46],
            in2 := "Data_block_1".data_baru1[47],
            in3 := 2.0,
            out => "Data_block_1".data_lama1);
   END_IF;
   IF #_w1 AND ("Data_block_1".counter_datasuhu = 95) THEN
       "Data_block_1".data_lama1 := "Data_block_1".data_baru1[47];
   END_IF;
   IF #_w1 AND ("Data_block_1".counter_datasuhu = 96) THEN
       CALC(in1 := "Data_block_1".data_baru1[47],
            in2 := "Data_block_1".data_baru1[48],
            in3 := 2.0,
            out => "Data_block_1".data_lama1);
   END_IF;
   IF #_w1 AND ("Data_block_1".counter_datasuhu = 97) THEN
       "Data_block_1".data_lama1 := "Data_block_1".data_baru1[48];
   END_IF;
   IF #_w1 AND ("Data_block_1".counter_datasuhu = 98) THEN
       CALC(in1 := "Data_block_1".data_baru1[48],
            in2 := "Data_block_1".data_baru1[49],
            in3 := 2.0,
            out => "Data_block_1".data_lama1);
   END_IF;
   IF #_w1 AND ("Data_block_1".counter_datasuhu = 99) THEN
       "Data_block_1".data_lama1 := "Data_block_1".data_baru1[49];
   END_IF;
   IF #_w1 AND ("Data_block_1".counter_datasuhu = 100) THEN
       CALC(in1 := "Data_block_1".data_baru1[49],
            in2 := "Data_block_1".data_baru1[50],
            in3 := 2.0,
            out => "Data_block_1".data_lama1);
   END_IF;
END_REGION

REGION Network 28: Menentukan Nilai Tengah (Kiri)
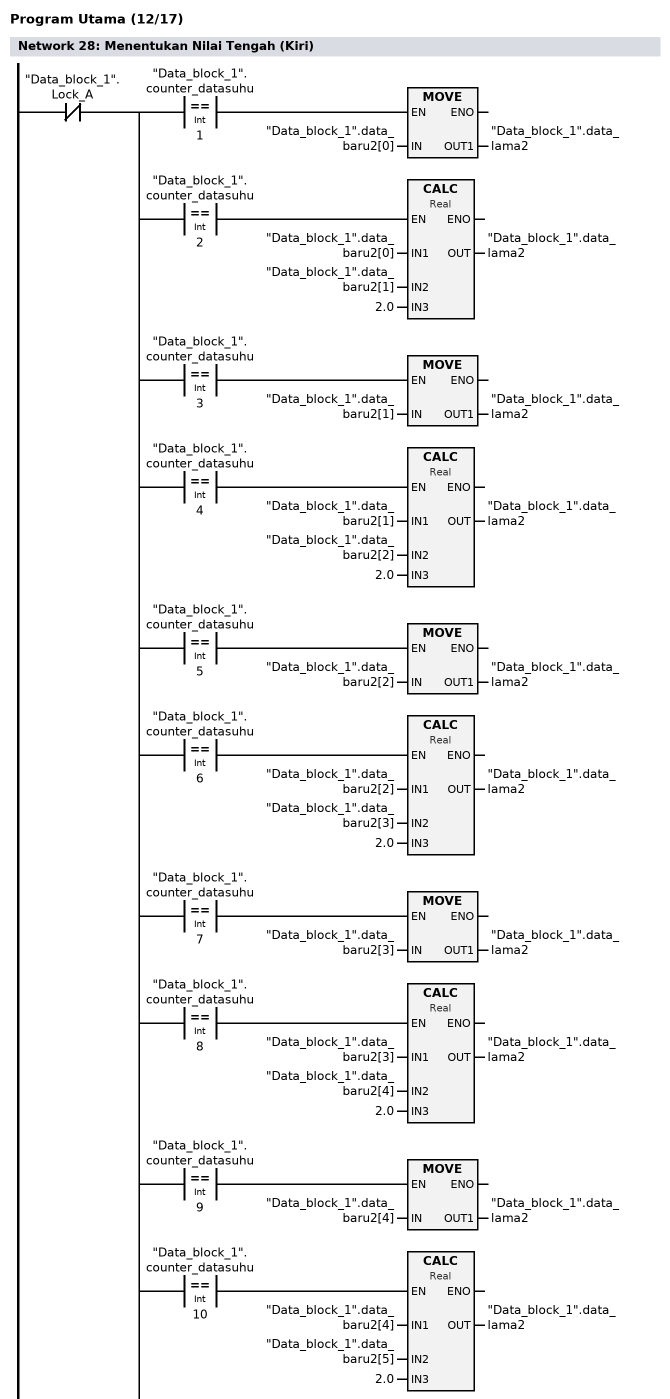
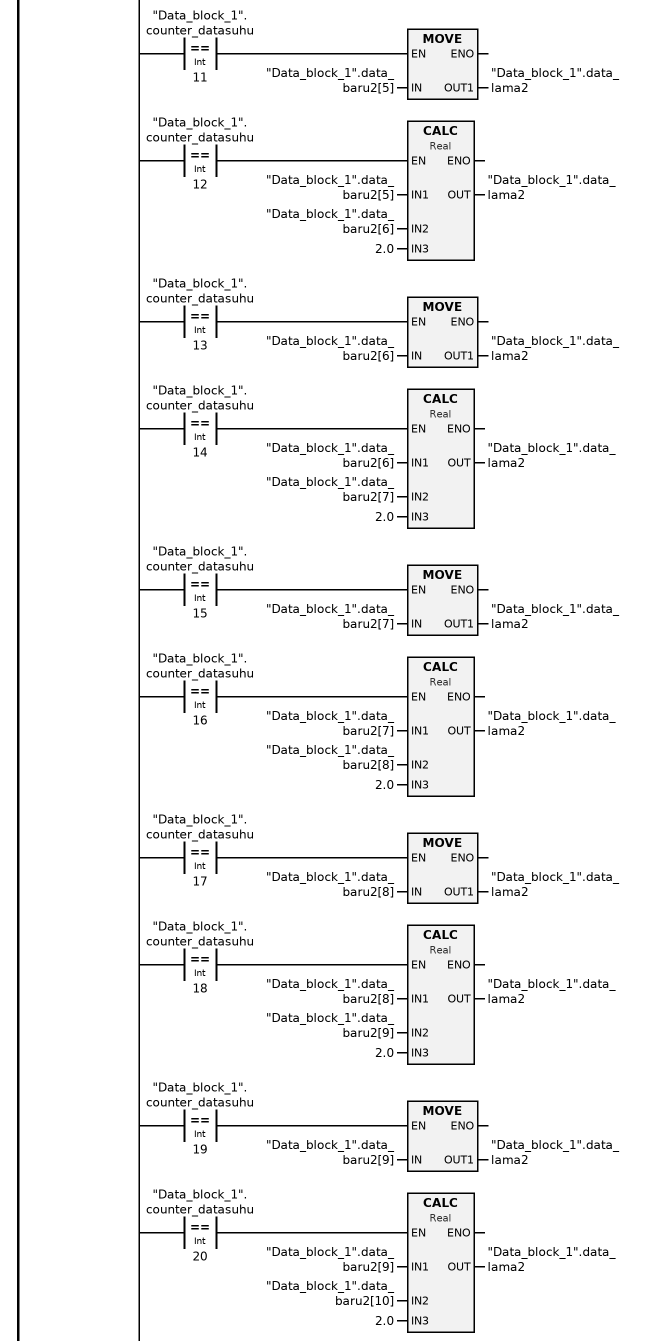
